// call fb cyclic
fbHoming.bCalibrationCam := bCalibrationCam;	
fbHoming.BufferMode := stHomingPrm.eBufferMode;
fbHoming.HomingMode := stHomingPrm.eHomingMode;
fbHoming.Options := stHomingPrm.stOptions;
fbHoming.Position := stHomingPrm.fPosition;
fbHoming(Axis := fbAxisRef);

// FB diagnostic and reset 
IF fbHoming.Execute AND NOT fbHoming.Busy THEN
	IF fbHoming.Error THEN
		nErrorId := fbHoming.ErrorID;
		M_SetLocalErrorS('Error axis homing: ErrId: ', TO_STRING(nErrorId));
	END_IF
	fbHoming.Execute := FALSE;
END_IF
		
// return if not in homing
IF eCommandExecute <> E_MotionCommand.eMotionCommand_home THEN
	RETURN;
END_IF

//aSClearText[0] := 'Antrieb GRST';	
//aSClearText := F_GetTranslatedTxtEx("engine home position", eLanguage);	
IF NOT fbHoming.Busy THEN
	fbHoming(Axis := fbAxisRef, Execute := TRUE);
	eCommandExecute := E_MotionCommand.eMotionCommand_none;
END_IF
END_ACTION

METHOD PRIVATE WfInitPositionOffset : BOOL
VAR_INPUT
END_VAR
VAR_INST
	fbAdsWriteOffset			:ADSWRITE;
	iStepSetPosOffset			:INT;
END_VAR


CASE iStepSetPosOffset OF
	
	0:
		// warte auf Trigger
		IF bStartInitPosOffset THEN
			// Position offset set
			bSetPositionOffsetDone := FALSE;
			// Current position offset value
			fCurrentPositionOffset := 0;			
			iStepSetPosOffset := 5;
		END_IF	
		
	5:
		IF fbAxisRef.NcToPlc.AxisId > 0 THEN
			iStepSetPosOffset := 6;
		ELSE
			M_SetLocalErrorEx(CONST.stTextListGlobal.stText_Comp.stText_Axis_FbError, F_CreateDynText("No Nc.AxisId!", 0));
		END_IF

	6:
		IF NOT Operational THEN
			iStepSetPosOffset := 10;
		ELSE
			M_SetLocalErrorEx(CONST.stTextListGlobal.stText_Comp.stText_Axis_FbError, F_CreateDynText("Axis is Operational. Please switch off axis!", 0));
		END_IF

	10:
		fbAdsWriteOffset.IDXGRP := 16#5000 + fbAxisRef.NcToPlc.AxisId;        (* Ind.Gr. f. AxisPara *)
		fbAdsWriteOffset.IDXOFFS := 16#7;
		fbAdsWriteOffset.LEN:= SIZEOF(fPosOffsetValToSet);
		fbAdsWriteOffset.SRCADDR:= ADR(fPosOffsetValToSet);
		fbAdsWriteOffset.WRITE:= TRUE;
		iStepSetPosOffset := 15;
   
    15:
        // 'wait until offset-parameter is handed over';
        IF NOT fbAdsWriteOffset.BUSY THEN
            IF fbAdsWriteOffset.ERRID = 0 THEN
				// Position offset set
				bSetPositionOffsetDone := TRUE;
				// Current position offset value
				fCurrentPositionOffset := fPosOffsetValToSet;
                iStepSetPosOffset := 100;
            ELSE
                M_SetLocalErrorEx(CONST.stTextListGlobal.stText_Comp.stText_Axis_FbError, F_CreateDynText("Error writing offset to NC.", 0));
				iStepSetPosOffset := 100;
            END_IF
        END_IF	
		

		// finish
	100:
		fbAdsWriteOffset.WRITE:= FALSE;
		bStartInitPosOffset := FALSE; // Finish
		fPosOffsetValToSet := 0;
		iStepSetPosOffset := 0;

END_CASE

fbAdsWriteOffset.PORT := 500;
fbAdsWriteOffset();
END_METHOD

ACTION WfJog:

/// Workflow jog axis

// call fb cyclic
fbjog.JogBackwards := stJogPrm.bJogBackwards AND Operational;
fbjog.JogForward := stJogPrm.bJogForward AND Operational;
fbjog.Acceleration := stJogPrm.fAcceleration;
fbjog.Deceleration := stJogPrm.fDeceleration;
fbjog.Jerk := stJogPrm.fJerk;
fbjog.Mode := stJogPrm.eMode;
fbjog.Position := stJogPrm.fPosition;
fbjog.Velocity := stJogPrm.fVelocity;
fbjog(Axis := fbAxisRef);

// reset jog F/B each cycle (stop's axis if Jog/JogEx method isn't called anymore)
stJogPrm.bJogBackwards := FALSE;
stJogPrm.bJogForward := FALSE;

// return if not in jog
IF eCommandExecute <> E_MotionCommand.eMotionCommand_jog THEN
	RETURN;
END_IF

// case of jog error
IF fbjog.Error  THEN
	nErrorId := fbjog.ErrorID;
	M_SetLocalErrorS('Error axis jogging: ErrId: ', TO_STRING(nErrorId));
END_IF		

eCommandExecute := E_MotionCommand.eMotionCommand_none;
END_ACTION

ACTION WfJogAcc:

/// Workflow jog axis acc

// call fb's cyclic
//fbJogAcc.Direction := MC_Current_Direction;
//IF stJogAccPrm.bJogForward OR stJogAccPrm.bJogBackwards THEN
fbJogAcc.Direction := SEL(stJogAccPrm.bJogForward, MC_Negative_Direction, MC_Positive_Direction);	
//END_IF
fbJogAcc.Acceleration := stJogAccPrm.fAcceleration;
fbJogAcc.Deceleration := stJogAccPrm.fDeceleration;
fbJogAcc.Jerk := stJogAccPrm.fJerk;
fbJogAcc.BufferMode := stJogAccPrm.eBufferMode;
fbJogAcc.Options := stJogAccPrm.stOptions;
fbJogAcc(Axis := fbAxisRef);

// FB diagnostic and reset 
IF fbJogAcc.Execute AND (NOT fbJogAcc.Busy OR fbJogAcc.InVelocity) THEN
	IF fbJogAcc.Error THEN
		nErrorId := fbJogAcc.ErrorID;
		M_SetLocalErrorS('Error axis jogging acceleration: ErrId: ', TO_STRING(nErrorId));
	END_IF
	fbJogAcc.Velocity := 0;
	fbJogAcc.Execute := FALSE;
END_IF

// measure jog time to capture speed at the according ramp positon
tonJogAcc.IN := stJogAccPrm.bJogForward OR stJogAccPrm.bJogBackwards;
tonJogAcc.PT := stJogAccPrm.tAccTime;
tonJogAcc();

// reset jog F/B each cycle (stop's axis if Jog/JogEx method isn't called anymore)
stJogAccPrm.bJogBackwards := FALSE;
stJogAccPrm.bJogForward := FALSE;

IF eCommandExecute <> E_MotionCommand.eMotionCommand_jogAcc THEN
	RETURN;
END_IF

// halt axis if jogAcc timer is disabled
IF NOT tonJogAcc.IN THEN
	fbJogAcc.Velocity := 0;
	eCommandExecute := E_MotionCommand.eMotionCommand_none;
	stHaltPrm.eBufferMode := MC_Aborting;
	stHaltPrm.fDeceleration := stJogAccPrm.fDeceleration;
	stHaltPrm.fJerk := stJogAccPrm.fJerk;
	stHaltPrm.stOptions := stJogAccPrm.stOptions;
	THIS^.HaltEx(stHaltPrm);	
END_IF

//aSClearText[0] := Concat2x('Antrieb Tippen Beschleunigung, Geschwindigkeit: ', LREAL_TO_STRING(fbJogAcc.Velocity));
//aSClearText := Concat2x(F_GetTranslatedTxtLib('type engine acceleration, acceleration: ', eLanguage), LREAL_TO_STRING(fbJogAcc.Velocity));
IF fbJogAcc.Velocity < stJogAccPrm.fFastSpeed AND NOT fbJogAcc.Busy THEN
	// ramp = Kx + d
	fbJogAcc.Velocity := (TIME_TO_LREAL(tonJogAcc.ET) * ((stJogAccPrm.fFastSpeed - stJogAccPrm.fSlowSpeed)/TIME_TO_LREAL(tonJogAcc.PT))) + stJogAccPrm.fSlowSpeed;
	// limit speed	
	fbJogAcc.Velocity := LIMIT(stJogAccPrm.fSlowSpeed, fbJogAcc.Velocity, stJogAccPrm.fFastSpeed);
	fbJogAcc(Axis := fbAxisRef, Execute := TRUE);	
END_IF
END_ACTION

ACTION WfMovAbs:

/// Workflow move axis abs

// call fb's cyclic
fbMovAbs1.Position := stMovAbsPrm.fPosition;
fbMovAbs1.Velocity := stMovAbsPrm.fVelocity;
fbMovAbs1.Acceleration := stMovAbsPrm.fAcceleration;
fbMovAbs1.Deceleration := stMovAbsPrm.fDeceleration;
fbMovAbs1.Jerk := stMovAbsPrm.fJerk;
fbMovAbs1.BufferMode := stMovAbsPrm.eBufferMode;
fbMovAbs1.Options := stMovAbsPrm.stOptions;
fbMovAbs1(Axis := fbAxisRef);

fbMovAbs2.Position := stMovAbsPrm.fPosition;
fbMovAbs2.Velocity := stMovAbsPrm.fVelocity;
fbMovAbs2.Acceleration := stMovAbsPrm.fAcceleration;
fbMovAbs2.Deceleration := stMovAbsPrm.fDeceleration;
fbMovAbs2.Jerk := stMovAbsPrm.fJerk;
fbMovAbs2.BufferMode := stMovAbsPrm.eBufferMode;
fbMovAbs2.Options := stMovAbsPrm.stOptions;
fbMovAbs2(Axis := fbAxisRef);

bMovAbsRdy := NOT (fbMovAbs1.Busy AND fbMovAbs2.Busy);

// FB diagnostic and reset 
IF fbMovAbs1.Execute AND NOT fbMovAbs1.Busy THEN
	IF fbMovAbs1.Error AND (fbMovAbs1.ErrorID <> 17022) THEN
		nErrorId := fbMovAbs1.ErrorID;
		M_SetLocalErrorS('engine positioning absolut (FB1): ErrId: ', TO_STRING(nErrorId));
	END_IF
	fbMovAbs1.Execute := FALSE;
END_IF
IF fbMovAbs2.Execute AND NOT fbMovAbs2.Busy THEN
	IF fbMovAbs2.Error AND (fbMovAbs2.ErrorID <> 17022) THEN
		nErrorId := fbMovAbs2.ErrorID;
		M_SetLocalErrorS('engine positioning absolut (FB2): ErrId: ', TO_STRING(nErrorId));
	END_IF
	fbMovAbs2.Execute := FALSE;
END_IF

// return if not in move abs
IF eCommandExecute <> E_MotionCommand.eMotionCommand_moveAbs THEN
	RETURN;
END_IF

//aSClearText[0] := 'Antrieb Positionierung Absolut';	
//aSClearText := F_GetTranslatedTxtLib('engine positioning absolut', eLanguage);
IF NOT fbMovAbs1.Busy THEN
	fbMovAbs1(Axis := fbAxisRef, Execute := TRUE);
	eCommandExecute := E_MotionCommand.eMotionCommand_none;
ELSIF NOT fbMovAbs2.Busy THEN
	fbMovAbs2(Axis := fbAxisRef, Execute := TRUE);
	eCommandExecute := E_MotionCommand.eMotionCommand_none;
ELSE
	nErrorId := 0;
	M_SetLocalError(F_CreateDynText("engine positioning absolut. No component ready", 0));
END_IF
END_ACTION

ACTION WfMovAdd:

/// Workflow move axis add

// call fb's cyclic
fbMovAdd1.Distance := stMovAddPrm.fDistance;
fbMovAdd1.Velocity := stMovAddPrm.fVelocity;
fbMovAdd1.Acceleration := stMovAddPrm.fAcceleration;
fbMovAdd1.Deceleration := stMovAddPrm.fDeceleration;
fbMovAdd1.Jerk := stMovAddPrm.fJerk;
fbMovAdd1.BufferMode := stMovAddPrm.eBufferMode;
fbMovAdd1.Options := stMovAddPrm.stOptions;
fbMovAdd1(Axis := fbAxisRef);

fbMovAdd2.Distance := stMovAddPrm.fDistance;
fbMovAdd2.Velocity := stMovAddPrm.fVelocity;
fbMovAdd2.Acceleration := stMovAddPrm.fAcceleration;
fbMovAdd2.Deceleration := stMovAddPrm.fDeceleration;
fbMovAdd2.Jerk := stMovAddPrm.fJerk;
fbMovAdd2.BufferMode := stMovAddPrm.eBufferMode;
fbMovAdd2.Options := stMovAddPrm.stOptions;
fbMovAdd2(Axis := fbAxisRef);

// FB diagnostic and reset 
IF fbMovAdd1.Execute AND NOT fbMovAdd1.Busy THEN
	IF fbMovAdd1.Error AND (fbMovAdd1.ErrorID <> 17022) THEN
		nErrorId := fbMovAdd1.ErrorID;
		M_SetLocalErrorS('engine positioning additive (FB1): ErrId: ', TO_STRING(nErrorId));
	END_IF
	fbMovAdd1.Execute := FALSE;
END_IF
IF fbMovAdd2.Execute AND NOT fbMovAdd2.Busy THEN
	IF fbMovAdd2.Error AND (fbMovAdd2.ErrorID <> 17022) THEN
		nErrorId := fbMovAdd2.ErrorID;
		M_SetLocalErrorS('engine positioning additive (FB2): ErrId: ', TO_STRING(nErrorId));
	END_IF
	fbMovAdd2.Execute := FALSE;
END_IF

// return if not in move add
IF eCommandExecute <> E_MotionCommand.eMotionCommand_moveAdd THEN
	RETURN;
END_IF

//aSClearText := F_GetTranslatedTxtLib('engine positioning additive', eLanguage);
IF NOT fbMovAdd1.Busy THEN
	fbMovAdd1(Axis := fbAxisRef, Execute := TRUE);
	eCommandExecute := E_MotionCommand.eMotionCommand_none;	
ELSIF NOT fbMovAdd2.Busy THEN
	fbMovAdd2(Axis := fbAxisRef, Execute := TRUE);
	eCommandExecute := E_MotionCommand.eMotionCommand_none;	
ELSE
	nErrorId := 0;
	M_SetLocalError(F_CreateDynText("engine positioning additive. No component ready", 0));
END_IF
END_ACTION

ACTION WfMovMod:

/// Workflow move axis mod

// call fb's cyclic
fbMovMod1.Position := stMovModPrm.fPosition;
fbMovMod1.Direction := stMovModPrm.eDirection;
fbMovMod1.Velocity := stMovModPrm.fVelocity;
fbMovMod1.Acceleration := stMovModPrm.fAcceleration;
fbMovMod1.Deceleration := stMovModPrm.fDeceleration;
fbMovMod1.Jerk := stMovModPrm.fJerk;
fbMovMod1.BufferMode := stMovModPrm.eBufferMode;
fbMovMod1.Options := stMovModPrm.stOptions;
fbMovMod1(Axis := fbAxisRef);

fbMovMod2.Position := stMovModPrm.fPosition;
fbMovMod2.Direction := stMovModPrm.eDirection;
fbMovMod2.Velocity := stMovModPrm.fVelocity;
fbMovMod2.Acceleration := stMovModPrm.fAcceleration;
fbMovMod2.Deceleration := stMovModPrm.fDeceleration;
fbMovMod2.Jerk := stMovModPrm.fJerk;
fbMovMod2.BufferMode := stMovModPrm.eBufferMode;
fbMovMod2.Options := stMovModPrm.stOptions;
fbMovMod2(Axis := fbAxisRef);

// FB diagnostic and reset 
IF fbMovMod1.Execute AND NOT fbMovMod1.Busy THEN
	IF fbMovMod1.Error AND (fbMovMod1.ErrorID <> 17022) THEN
		nErrorId := fbMovMod1.ErrorID;
		M_SetLocalErrorS('engine positioning modulo (FB1): ErrId: ', TO_STRING(nErrorId));
	END_IF
	fbMovMod1.Execute := FALSE;
END_IF
IF fbMovMod2.Execute AND NOT fbMovMod2.Busy THEN
	IF fbMovMod2.Error AND (fbMovMod2.ErrorID <> 17022) THEN
		nErrorId := fbMovMod2.ErrorID;
		M_SetLocalErrorS('engine positioning modulo (FB2): ErrId: ', TO_STRING(nErrorId));
	END_IF
	fbMovMod2.Execute := FALSE;
END_IF

// return if not in move rel
IF eCommandExecute <> E_MotionCommand.eMotionCommand_moveMod THEN
	RETURN;
END_IF

//aSClearText[0] := 'Antrieb Positionierung Modulo';	
//aSClearText := F_GetTranslatedTxtLib('engine positioning modulo', eLanguage);	
IF NOT fbMovMod1.Busy THEN
	fbMovMod1(Axis := fbAxisRef, Execute := TRUE);
	eCommandExecute := E_MotionCommand.eMotionCommand_none;
ELSIF NOT fbMovMod2.Busy THEN
	fbMovMod2(Axis := fbAxisRef, Execute := TRUE);
	eCommandExecute := E_MotionCommand.eMotionCommand_none;
ELSE
	nErrorId := 0;
	M_SetLocalError(F_CreateDynText("engine positioning modulo. No component ready", 0));
END_IF
END_ACTION

ACTION WfMovRel:

/// Workflow move axis rel

// call fb's cyclic
fbMovRel1.Distance := stMovRelPrm.fDistance;
fbMovRel1.Velocity := stMovRelPrm.fVelocity;
fbMovRel1.Acceleration := stMovRelPrm.fAcceleration;
fbMovRel1.Deceleration := stMovRelPrm.fDeceleration;
fbMovRel1.Jerk := stMovRelPrm.fJerk;
fbMovRel1.BufferMode := stMovRelPrm.eBufferMode;
fbMovRel1.Options := stMovRelPrm.stOptions;
fbMovRel1(Axis := fbAxisRef);

fbMovRel2.Distance := stMovRelPrm.fDistance;
fbMovRel2.Velocity := stMovRelPrm.fVelocity;
fbMovRel2.Acceleration := stMovRelPrm.fAcceleration;
fbMovRel2.Deceleration := stMovRelPrm.fDeceleration;
fbMovRel2.Jerk := stMovRelPrm.fJerk;
fbMovRel2.BufferMode := stMovRelPrm.eBufferMode;
fbMovRel2.Options := stMovRelPrm.stOptions;
fbMovRel2(Axis := fbAxisRef);

// FB diagnostic and reset 
IF fbMovRel1.Execute AND NOT fbMovRel1.Busy THEN
	IF fbMovRel1.Error AND (fbMovRel1.ErrorID <> 17022) THEN
		nErrorId := fbMovRel1.ErrorID;
		M_SetLocalErrorS('engine positioning relativ (FB1): ErrId: ', TO_STRING(nErrorId));
	END_IF
	fbMovRel1.Execute := FALSE;
END_IF
IF fbMovRel2.Execute AND NOT fbMovRel2.Busy THEN
	IF fbMovRel2.Error AND (fbMovRel2.ErrorID <> 17022) THEN
		nErrorId := fbMovRel2.ErrorID;
		M_SetLocalErrorS('engine positioning relativ (FB2): ErrId: ', TO_STRING(nErrorId));
	END_IF
	fbMovRel2.Execute := FALSE;
END_IF

// return if not in move rel
IF eCommandExecute <> E_MotionCommand.eMotionCommand_moveRel THEN
	RETURN;
END_IF

//aSClearText := F_GetTranslatedTxtLib('engine positioning relativ', eLanguage);
IF NOT fbMovRel1.Busy THEN
	fbMovRel1(Axis := fbAxisRef, Execute := TRUE);
	eCommandExecute := E_MotionCommand.eMotionCommand_none;	
ELSIF NOT fbMovRel2.Busy THEN
	fbMovRel2(Axis := fbAxisRef, Execute := TRUE);
	eCommandExecute := E_MotionCommand.eMotionCommand_none;	
ELSE
	nErrorId := 0;
	M_SetLocalError(F_CreateDynText("engine positioning relativ. No component ready", 0));
END_IF
END_ACTION

ACTION WfMovVel:

/// Workflow move axis vel

// call fb's cyclic
fbMovVel1.Velocity := stMovVelPrm.fVelocity;
fbMovVel1.Direction := stMovVelPrm.eDirection;
fbMovVel1.Acceleration := stMovVelPrm.fAcceleration;
fbMovVel1.Deceleration := stMovVelPrm.fDeceleration;
fbMovVel1.Jerk := stMovVelPrm.fJerk;
fbMovVel1.BufferMode := stMovVelPrm.eBufferMode;
fbMovVel1.Options := stMovVelPrm.stOptions;
fbMovVel1(Axis := fbAxisRef);

fbMovVel2.Velocity := stMovVelPrm.fVelocity;
fbMovVel2.Direction := stMovVelPrm.eDirection;
fbMovVel2.Acceleration := stMovVelPrm.fAcceleration;
fbMovVel2.Deceleration := stMovVelPrm.fDeceleration;
fbMovVel2.Jerk := stMovVelPrm.fJerk;
fbMovVel2.BufferMode := stMovVelPrm.eBufferMode;
fbMovVel2.Options := stMovVelPrm.stOptions;
fbMovVel2(Axis := fbAxisRef);

// FB diagnostic and reset 
IF fbMovVel1.Execute AND NOT fbMovVel1.Busy THEN
	IF fbMovVel1.Error AND (fbMovVel1.ErrorID <> 17022) THEN
		nErrorId := fbMovVel1.ErrorID;
		M_SetLocalErrorS('engine constant velocity (FB1): ErrId: ', TO_STRING(nErrorId));
	END_IF
	fbMovVel1.Execute := FALSE;
END_IF
IF fbMovVel2.Execute AND NOT fbMovVel2.Busy THEN
	IF fbMovVel2.Error AND (fbMovVel2.ErrorID <> 17022) THEN
		nErrorId := fbMovVel2.ErrorID;
		M_SetLocalErrorS('engine constant velocity (FB2): ErrId: ', TO_STRING(nErrorId));
	END_IF
	fbMovVel2.Execute := FALSE;
END_IF

// return if other command active
IF eCommandExecute <> E_MotionCommand.eMotionCommand_moveVel THEN
	RETURN;
END_IF

//aSClearText[0] := 'Antrieb Konstante Geschwindigkeit';
//aSClearText := F_GetTranslatedTxtLib('engine constant velocity', eLanguage);				
IF NOT fbMovVel1.Busy THEN
	fbMovVel1(Axis := fbAxisRef, Execute := TRUE);
	eCommandExecute := E_MotionCommand.eMotionCommand_none;
ELSIF NOT fbMovVel2.Busy THEN
	fbMovVel2(Axis := fbAxisRef, Execute := TRUE);
	eCommandExecute := E_MotionCommand.eMotionCommand_none;
ELSE
	nErrorId := 0;
	M_SetLocalError(F_CreateDynText("engine constant velocity. No Component ready", 0));
END_IF
END_ACTION

ACTION WfPower:

/// Workflow power axis

tonAutoPowerOff(IN := bEnable AND bEnableAutoPowerOff AND fbAxisRef.Status.NotMoving AND NOT fbAxisRef.Status.Error AND 
					  (eCommandRequest = eMotionCommand_none OR eCommandRequest = eMotionCommand_reset OR eCommandRequest = eMotionCommand_setPos) AND
					  (eCommandExecute = eMotionCommand_none OR eCommandExecute = eMotionCommand_reset OR eCommandExecute = eMotionCommand_setPos),
				PT := stDefaultPrm.stGeneralPrm.tAutoPowerOffDelay);

tonEnable(IN:=bEnable,PT := tEnableTime);
				
fbPower.Enable := tonEnable.Q AND NOT tonAutoPowerOff.Q;
fbPower.Enable_Negative := bEnableNeg;
fbPower.Enable_Positive := bEnablePos;
fbPower.Override := SEL(bHoldActiv,fSetOverride,0);
fbPower(BufferMode := MC_Aborting, Axis := fbAxisRef);

// ext. fan control
IF stIn.iMotorTemperature >= stDefaultPrm.stGeneralPrm.iExtFanThreshold THEN
	stOut.bExternalFan := TRUE;
ELSIF stIn.iMotorTemperature < (stDefaultPrm.stGeneralPrm.iExtFanThreshold - 50) THEN // hysteresis 5°C
	stOut.bExternalFan := FALSE;
END_IF

posPowerError(CLK := eState <> E_ComponentState.eComponentState_error AND fbPower.Error);
IF posPowerError.Q THEN
	nErrorId := fbPower.ErrorID;
	M_SetLocalErrorS('Axis power error: ErrId: ', TO_STRING(nErrorId));
END_IF
END_ACTION

ACTION WfReset:

/// Workflow resetting

// call FB cyclic
fbReset(Axis:= fbAxisRef);

// FB diagnostic and reset 
IF fbReset.Execute AND NOT fbReset.Busy THEN
	IF fbReset.Error THEN			
		nErrorId := fbReset.ErrorID;
		M_SetLocalErrorS('Error on engine reset: ErrId: ', TO_STRING(nErrorId));
	END_IF
	fbReset.Execute := FALSE;
END_IF

// force MC reset
IF eCommandExecute = eMotionCommand_resetMc THEN
	//aSClearText[0] := 'Start Antrieb MC Reset';
	//aSClearText := F_GetTranslatedTxtEx("Start engine MC reset", eLanguage);
	IF NOT fbReset.Busy THEN
		fbReset(Axis := fbAxisRef, Execute := TRUE);
		eCommandExecute := E_MotionCommand.eMotionCommand_none;
	END_IF
END_IF

// return if other command active
IF eCommandExecute <> E_MotionCommand.eMotionCommand_reset THEN
	RETURN;
END_IF

IF eAxisType = E_AxisType.AX5xxx THEN
	// reset ax5000
	//aSClearText := F_GetTranslatedTxtEx("Start engine reset", eLanguage);
	IF NOT fbAX5xxxDiag.Busy THEN
		fbAX5xxxDiag.Reset := fbAxisRef.Status.Error;
		eCommandExecute := E_MotionCommand.eMotionCommand_none;
		eState := E_ComponentState.eComponentState_ready;
	END_IF

// Bosch Indradrive
ELSIF eAxisType = E_AxisType.Bosch_IndradriveEc THEN
	// reset indradrive
	//aSClearText := F_GetTranslatedTxtEx("Start engine reset", eLanguage);
	IF NOT fbIndraDrvDiag.bBusy THEN
		fbIndraDrvDiag.bReset := fbAxisRef.Status.Error;
		eCommandExecute := E_MotionCommand.eMotionCommand_none;
		eState := E_ComponentState.eComponentState_ready;
	END_IF

ELSE
	// reset sequence of default axis types
	//aSClearText := F_GetTranslatedTxtEx("Start engine reset", eLanguage);
	IF NOT fbReset.Busy THEN
		fbReset(Axis := fbAxisRef, Execute := fbAxisRef.Status.Error);
		eCommandExecute := E_MotionCommand.eMotionCommand_none;
		eState := E_ComponentState.eComponentState_ready;
	END_IF
END_IF
END_ACTION

ACTION WfSetPos:

/// Workflow set position

// call fb cyclic
fbSetPos.Position := stSetPosPrm.fPosition;
fbSetPos.Mode := stSetPosPrm.bMode;
fbSetPos.Options := stSetPosPrm.stOptions;
fbSetPos(Axis := fbAxisRef);

// FB diagnostic and reset 
IF fbSetPos.Execute AND NOT fbSetPos.Busy THEN
	IF fbSetPos.Error THEN			
		nErrorId := fbSetPos.ErrorID;
		M_SetLocalErrorS('Error set engine position: ErrId: ', TO_STRING(nErrorId));
	END_IF
	fbSetPos.Execute := FALSE;
END_IF

// return if other command active	
IF eCommandExecute <> E_MotionCommand.eMotionCommand_setPos THEN
	RETURN;
END_IF

//aSClearText := F_GetTranslatedTxtLib('Set engine position', eLanguage);		
IF NOT fbSetPos.Busy THEN
	fbSetPos(Axis := fbAxisRef, Execute := TRUE);
	eCommandExecute := E_MotionCommand.eMotionCommand_none;
END_IF
END_ACTION

ACTION WfSoE:
// SoE commands
CASE stSoE.eCmd OF
	
	E_SoECommand.eSoECommand_writeIndraDrvPos:
		CASE stSoE.nStep OF
			0:	
				stSoE.fRealValue := (stSoE.fRealValue * 10000);
				diTempVal := REAL_TO_DINT(stSoE.fRealValue);
				stSoE.fbSoEWrite(
					Axis    := fbAxisRef,
					Idn := S_0_IDN + 52, 				// S-0-0052, Referenzmaß 1
					Element := EC_SOE_ELEMENT_VALUE,
					pSrcBuf  := ADR(diTempVal),	// Position
					BufLen   := SIZEOF(diTempVal),
					//Password := Password,				// Password   : ST_SoE_String;
					Execute  := TRUE,
					Timeout  := DEFAULT_ADS_TIMEOUT);				
				IF NOT stSoE.fbSoEWrite.Busy THEN
					IF stSoE.fbSoEWrite.Error THEN
						eState := E_ComponentState.eComponentState_error;
						nErrorID := stSoE.fbSoEWrite.AdsErrId;
						M_SetLocalError(F_CreateDynText(TO_WSTRING(Concat4('SoEWrite error, AdsErrId: ', UINT_TO_STRING(stSoE.fbSoEWrite.AdsErrId), ', SercosErrId: ', UINT_TO_STRING(stSoE.fbSoEWrite.SercosErrId))), 0));
						stSoE.nStep := 0;
						stSoE.eCmd := E_SoECommand.eSoECommand_none;
					ELSE
						stSoE.nStep := 10;
					END_IF
					stSoE.fbSoEWrite(Axis := fbAxisRef, Execute := FALSE);
				END_IF
				
			10:	stSoE.fbSoECmd(
					Axis    := fbAxisRef,
					Execute := TRUE,
					Timeout := DEFAULT_ADS_TIMEOUT,
					Idn     := S_0_IDN + 447);			// C0300 Kommando Absolutmaß setzen		P_0_IDN + 12
				IF NOT stSoE.fbSoECmd.Busy THEN
					IF stSoE.fbSoECmd.Error THEN
						eState := E_ComponentState.eComponentState_error;
						nErrorID := stSoE.fbSoEWrite.AdsErrId;
						M_SetLocalError(F_CreateDynText(TO_WSTRING(Concat4('SoECmd error, AdsErrId: ', UINT_TO_STRING(stSoE.fbSoECmd.AdsErrId), ', SercosErrId: ', UINT_TO_STRING(stSoE.fbSoECmd.SercosErrId))), 0));
					END_IF
					stSoE.fbSoECmd(Axis := fbAxisRef, Execute := FALSE);
					stSoE.nStep := 0;
					stSoE.eCmd := E_SoECommand.eSoECommand_none;
				END_IF
				
		END_CASE
		
END_CASE
END_ACTION

ACTION WfStop:

/// Workflow stopping

// call fb cyclic
fbStop.Deceleration := stStopPrm.fDeceleration;
fbStop.Jerk := stStopPrm.fJerk;
fbStop.Options := stStopPrm.stOptions;
fbStop(Axis := fbAxisRef);

// FB diagnostic and reset
IF fbStop.Execute THEN
	IF fbStop.Error THEN			
		nErrorId := fbStop.ErrorID;
		M_SetLocalErrorS('Error stopping axis: ErrId: ', TO_STRING(nErrorId));
	END_IF
	fbStop.Execute := FALSE;
END_IF

// return if other command active
IF eCommandExecute <> E_MotionCommand.eMotionCommand_stop THEN
	RETURN;
END_IF

//aSClearText[0] := 'Antrieb Stoppen';
//aSClearText := F_GetTranslatedTxtLib('stop the engine ', eLanguage);
fbStop(Axis := fbAxisRef, Execute := TRUE);

// stop command is not auto reset -> ext. reset needed!

//IF fbAxisRef.Status.StandStill AND fbStop.Done AND NOT fbStop.Busy THEN
	eCommandExecute := E_MotionCommand.eMotionCommand_none;
//END_IF
END_ACTION

ACTION WfTorqCtrl:

/// Workflow torque control
stTorqCtrlPrm.stOptions.ManualTorqueStartValue := fbAxisRef.NcToPlc.ActTorque;
stTorqCtrlPrm.stOptions.EnableManualTorqueStartValue := TRUE;

// call fb cyclic
fbTorqueControl.Torque := stTorqCtrlPrm.fTorque;
fbTorqueControl.TorqueRamp := stTorqCtrlPrm.fTorqueRamp;
fbTorqueControl.VelocityLimitHigh := stTorqCtrlPrm.fVelocityLimitHigh;
fbTorqueControl.VelocityLimitLow := stTorqCtrlPrm.fVelocityLimitLow;
fbTorqueControl.ContinuousUpdate := stTorqCtrlPrm.bContinuousUpdate;
fbTorqueControl.Relative := stTorqCtrlPrm.bRelative;
fbTorqueControl.BufferMode := stTorqCtrlPrm.eBufferMode;
fbTorqueControl.Options := stTorqCtrlPrm.stOptions;
fbTorqueControl(Axis := fbAxisRef);

// FB diagnostic and reset 
IF fbTorqueControl.Execute AND NOT fbTorqueControl.Busy THEN
	IF fbTorqueControl.Error AND (fbTorqueControl.ErrorID <> 17022) THEN
		nErrorId := fbTorqueControl.ErrorID;
		M_SetLocalErrorS('engine torque control: ErrId: ', TO_STRING(nErrorId));
	END_IF
	fbTorqueControl.Execute := FALSE;
END_IF

// return if not in torque control
IF eCommandExecute <> E_MotionCommand.eMotionCommand_torqCtrl THEN
	RETURN;
END_IF

//IF NOT fbTorqueControl.Busy THEN
	fbTorqueControl(Axis := fbAxisRef, ContinuousUpdate := stTorqCtrlPrm.bContinuousUpdate, Execute := TRUE);
	eCommandExecute := E_MotionCommand.eMotionCommand_none;
//ELSE
//	nErrorId := 0;
//	M_SetLocalError(F_CreateDynText("engine torque control. Component not ready", 0));
//END_IF
END_ACTION

END_FUNCTION_BLOCK

// ---- POUs/MAIN_Fast.TcPOU
PROGRAM MAIN_Fast
VAR_INPUT
END_VAR
VAR
END_VAR
VAR_OUTPUT	
END_VAR

// fast stuff here..

fbModul001.M_Fast();

END_PROGRAM

// ---- POUs/HMI/Provider/HwHmi/FB_HMI_PROVIDER_HW.TcPOU
FUNCTION_BLOCK FB_HMI_PROVIDER_HW EXTENDS FB_HMI_PROVIDER_BASE
VAR
	stIn		: REFERENCE TO HMI_PROVIDER_HW_IN;
	stOut		: REFERENCE TO HMI_PROVIDER_HW_OUT;
	bLedTest	: BOOL;
	
	nSelStation : E_Station;
	bAlternativ : BOOL;	
	bJog : BOOL;
	bSpeed : BOOL;

	
END_VAR

METHOD M_EuchnerToPLC : BOOL
VAR_INST		
	fbSelection				:FB_TON_RMTH;
	fbAlt					:FB_TON_RMTH;
	fbJog					:FB_TON_RMTH;
	fbSpeed					:FB_TON_RMTH;
	
	rtrigJog01				:R_TRIG;
	rtrigJog02				:R_TRIG;
	rtrigReset				:R_TRIG;
	
	nNewSelection			: INT;
END_VAR
fbSelection(IN := stIn.stP51A_S1HandBs.bSelect01 OR stIn.stP51A_S1HandBs.bSelect02 OR stIn.stP51A_S1HandBs.bSelect03 OR stIn.stP51A_S1HandBs.bSelect04 OR stIn.stP51A_S1HandBs.bSelect05 OR stIn.stP51A_S1HandBs.bSelect06 , PT:= T#50MS);	//Selection
fbAlt(IN := stIn.stP51A_S1HandBs.bAlt, PT:= T#50MS);	//Selection

fbJog(IN := stIn.stP51A_S1HandBs.bJog, PT:= T#50MS, Qr=> bJog);	//Selection
stIn.stSt010.bJog := stIn.stSt020.bJog := stIn.stSt030.bJog := stIn.stSt040.bJog := bJog;

fbSpeed(IN := stIn.stP51A_S1HandBs.bDistance, PT:= T#50MS);	//Selection

IF fbSpeed.Qr THEN
	bSpeed := NOT bSpeed;
END_IF

IF fbJog.Qr THEN
	bSpeed := FALSE;	
END_IF

stIn.stSt010.bSpeed := stIn.stSt020.bSpeed := stIn.stSt030.bSpeed := stIn.stSt040.bSpeed := bSpeed;

// Umschalten Station
IF fbSelection.Qr THEN
	bAlternativ := FALSE;
	IF stIn.stP51A_S1HandBs.bSelect01 THEN
		nNewSelection := E_Station.eStation_ST010_OvenA;
	ELSIF stIn.stP51A_S1HandBs.bSelect02 THEN
		nNewSelection := E_Station.eStation_ST020_OvenB;		
	ELSIF stIn.stP51A_S1HandBs.bSelect03 THEN
		nNewSelection := E_Station.eStation_ST030_Handling;		
	ELSIF stIn.stP51A_S1HandBs.bSelect04 THEN
		nNewSelection := E_Station.eStation_ST040_Storage;		
	ELSIF stIn.stP51A_S1HandBs.bSelect05 THEN
		nNewSelection := E_Station.eStation_ST050_Mould;		
	ELSIF stIn.stP51A_S1HandBs.bSelect06 THEN
		nNewSelection := E_Station.eStation_none;		
	END_IF
	
	IF nNewSelection = nSelStation THEN
		nSelStation := E_Station.eStation_none;
	ELSE
		nSelStation := nNewSelection;
	END_IF	
	
END_IF


// Umschalten auf Alternativ
IF fbAlt.Qr THEN
	bAlternativ := NOT bAlternativ;
END_IF
rtrigJog01(CLK := stIn.stP51A_S1HandBs.bLeft OR stIn.stP51A_S1HandBs.bRight);
rtrigJog02(CLK := stIn.stP51A_S1HandBs.bDown OR stIn.stP51A_S1HandBs.bUp);
rtrigReset(CLK := );

// Stationsfunktionen
CASE nSelStation OF
	

	eStation_none:  stIn.stM001.bQuit := stIn.stP51A_S1HandBs.bReset;

	
	eStation_ST010_OvenA: 	//stIn.stSt010.bManual := stIn.stP51A_S1HandBs.bReset;	
		stIn.stSt010.bQuit := stIn.stP51A_S1HandBs.bReset;

		// set up index	
		IF NOT bAlternativ THEN
			stOut.stP51A_S1HandBs.bLedLeft := TRUE;
			stOut.stP51A_S1HandBs.bLedRight := TRUE;	
			stIn.stSt010.bJogCh1Inside := stIn.stP51A_S1HandBs.bLeft;
	   		stIn.stSt010.bJogCh1Ouside := stIn.stP51A_S1HandBs.bRight;	
			IF rtrigJog01.Q THEN
				stIn.arrStStation[E_Station.eStation_ST010_OvenA].stManual.diSelectedObjectIndex := fbSt010OvenA.fbAxisCh1Ui.diObjectIndex;			
				bRequestManualControl := TRUE;
			END_IF					
		ELSE
			stOut.stP51A_S1HandBs.bLedLeft := TRUE;
			stOut.stP51A_S1HandBs.bLedRight := TRUE;
			stIn.stSt010.bJogCh2Inside := stIn.stP51A_S1HandBs.bLeft;
	   		stIn.stSt010.bJogCh2Ouside := stIn.stP51A_S1HandBs.bRight;	
			IF rtrigJog01.Q THEN
				stIn.arrStStation[E_Station.eStation_ST010_OvenA].stManual.diSelectedObjectIndex := fbSt010OvenA.fbAxisCh2Ui.diObjectIndex;
				bRequestManualControl := TRUE;
			END_IF
		END_IF
		
		stOut.stP51A_S1HandBs.bLedUp := TRUE;
		stOut.stP51A_S1HandBs.bLedDown := TRUE;
		stIn.stSt010.bJogUp := stIn.stP51A_S1HandBs.bUp;
		stIn.stSt010.bJogDown := stIn.stP51A_S1HandBs.bDown;
		IF rtrigJog02.Q THEN
			stIn.arrStStation[E_Station.eStation_ST010_OvenA].stManual.diSelectedObjectIndex := fbSt010OvenA.fbAxisUi.diObjectIndex;
			bRequestManualControl := TRUE;
		END_IF		
	
	eStation_ST020_OvenB: 	//stIn.stSt020.bManual := stIn.stP51A_S1HandBs.bReset;
		stIn.stSt020.bQuit := stIn.stP51A_S1HandBs.bReset;

		IF NOT bAlternativ THEN
			stOut.stP51A_S1HandBs.bLedLeft := TRUE;
			stOut.stP51A_S1HandBs.bLedRight := TRUE;	
			stIn.stSt020.bJogCh1Inside := stIn.stP51A_S1HandBs.bLeft;
	   		stIn.stSt020.bJogCh1Ouside := stIn.stP51A_S1HandBs.bRight;	
			IF rtrigJog01.Q THEN
				stIn.arrStStation[E_Station.eStation_ST020_OvenB].stManual.diSelectedObjectIndex := fbSt020OvenB.fbAxisCh1Ui.diObjectIndex;
				bRequestManualControl := TRUE;
			END_IF					
		ELSE
			stOut.stP51A_S1HandBs.bLedLeft := TRUE;
			stOut.stP51A_S1HandBs.bLedRight := TRUE;
			stIn.stSt020.bJogCh2Inside := stIn.stP51A_S1HandBs.bLeft;
	   		stIn.stSt020.bJogCh2Ouside := stIn.stP51A_S1HandBs.bRight;	
			IF rtrigJog01.Q THEN
				stIn.arrStStation[E_Station.eStation_ST020_OvenB].stManual.diSelectedObjectIndex := fbSt020OvenB.fbAxisCh2Ui.diObjectIndex;
				bRequestManualControl := TRUE;
			END_IF
		END_IF
		
		stOut.stP51A_S1HandBs.bLedUp := TRUE;
		stOut.stP51A_S1HandBs.bLedDown := TRUE;
		stIn.stSt020.bJogUp := stIn.stP51A_S1HandBs.bUp;
		stIn.stSt020.bJogDown := stIn.stP51A_S1HandBs.bDown;
		IF rtrigJog02.Q THEN
			stIn.arrStStation[E_Station.eStation_ST020_OvenB].stManual.diSelectedObjectIndex := fbSt020OvenB.fbAxisUi.diObjectIndex;
			bRequestManualControl := TRUE;
		END_IF	
	
	
	eStation_ST030_Handling: 	//stIn.stSt030.bManual := stIn.stP51A_S1HandBs.bReset;
		stIn.stSt030.bQuit := stIn.stP51A_S1HandBs.bReset;
	
		IF NOT bAlternativ THEN
			stOut.stP51A_S1HandBs.bLedLeft := TRUE;
			stOut.stP51A_S1HandBs.bLedRight := TRUE;
			stIn.stSt030.bJogXN := stIn.stP51A_S1HandBs.bLeft;
	   		stIn.stSt030.bJogXP := stIn.stP51A_S1HandBs.bRight;	
			IF rtrigJog01.Q THEN
				stIn.arrStStation[E_Station.eStation_ST030_Handling].stManual.diSelectedObjectIndex := fbSt030Handling.fbAxisXUi.diObjectIndex;
				bRequestManualControl := TRUE;
			END_IF	
			
			stOut.stP51A_S1HandBs.bLedUp := TRUE;
			stOut.stP51A_S1HandBs.bLedDown := TRUE;	
			stIn.stSt030.bJogYN := stIn.stP51A_S1HandBs.bDown;
	   		stIn.stSt030.bJogYP := stIn.stP51A_S1HandBs.bUp;
			IF rtrigJog02.Q THEN
				stIn.arrStStation[E_Station.eStation_ST030_Handling].stManual.diSelectedObjectIndex := fbSt030Handling.fbAxisYUi.diObjectIndex;
				bRequestManualControl := TRUE;
			END_IF	
	
		ELSE
			stOut.stP51A_S1HandBs.bLedLeft := TRUE;
			stOut.stP51A_S1HandBs.bLedRight := TRUE;
			stIn.stSt030.bJogZN := stIn.stP51A_S1HandBs.bLeft;
			stIn.stSt030.bJogZP := stIn.stP51A_S1HandBs.bRight;
			IF rtrigJog01.Q THEN
				stIn.arrStStation[E_Station.eStation_ST030_Handling].stManual.diSelectedObjectIndex := fbSt030Handling.fbAxisZUi.diObjectIndex;
				bRequestManualControl := TRUE;
			END_IF	
					
			stOut.stP51A_S1HandBs.bLedUp := FALSE;
			stOut.stP51A_S1HandBs.bLedDown := FALSE;
			
		END_IF		
		
	eStation_ST040_Storage: 	//stIn.stSt040.bManual := stIn.stP51A_S1HandBs.bReset;
		stIn.stSt040.bQuit := stIn.stP51A_S1HandBs.bReset;

		stOut.stP51A_S1HandBs.bLedLeft := FALSE;
		stOut.stP51A_S1HandBs.bLedRight := FALSE;	
	
		IF NOT bAlternativ THEN
			stOut.stP51A_S1HandBs.bLedUp := TRUE;
			stOut.stP51A_S1HandBs.bLedDown := TRUE;
			stIn.stSt040.bJog01Down := stIn.stP51A_S1HandBs.bDown;
	   		stIn.stSt040.bJog01Up := stIn.stP51A_S1HandBs.bUp;
			IF rtrigJog02.Q THEN
				stIn.arrStStation[E_Station.eStation_ST040_Storage].stManual.diSelectedObjectIndex := fbSt040Storage.fbAxis1Ui.diObjectIndex;
				bRequestManualControl := TRUE;
			END_IF					
		ELSE
			stOut.stP51A_S1HandBs.bLedUp := TRUE;
			stOut.stP51A_S1HandBs.bLedDown := TRUE;
			stIn.stSt040.bJog02Down := stIn.stP51A_S1HandBs.bDown;
	   		stIn.stSt040.bJog02Up := stIn.stP51A_S1HandBs.bUp;
			IF rtrigJog02.Q THEN
				stIn.arrStStation[E_Station.eStation_ST040_Storage].stManual.diSelectedObjectIndex := fbSt040Storage.fbAxis2Ui.diObjectIndex;
				bRequestManualControl := TRUE;
			END_IF
		END_IF
				

END_CASE




// chk control request, e.g.: watch for changes --> stIn..bJog.. (for continuous jog only!)
END_METHOD

METHOD PRIVATE M_HmiToPlc : BOOL
VAR_INST
	rtrigDoorP30A,
	rtrigDoorOpnP50A,
	rtrigDoorClsP50A,
	rtrigVorwHaerten,
	rtrigVorwAnlassen,
	rtrigAutoKorrS1,
	rtrigAutoKorrS2,
	rtrigAutoKorrS3,
	rtrigJog : R_TRIG;
END_VAR
/// general
stIn.stMain.stButton_Start.bClick := // stIn.stP10A_OvenA.bAutoOn OR	// Automatik Ein; LDT-GN, 1DI-NO, 1DO; +P30A-21SJ2
									 stIn.stP50A_Haupt.bAutoOn;				// Automatik Ein, LDT-GN, 1DI-NO, 1DO, BMK: +P50A-21SJ2

stIn.stMain.stButton_Stop.bClick := stIn.stP50A_Haupt.bAutoOff;// OR			// Automatik Aus, DT-RD, 1DI-NO, BMK: +P50A-21SJ3
									//stIn.stP10B_OvenB.bAutoOff;		// Automatik Aus; DT-RD, 1DI-NO; P10B-1SG2

//stIn.stMain.stButton_Home.bClick := stIn.bTaste_GRST;
//stIn.stMain.stButton_Step.bClick := stIn.bTaste_Tipp;
stIn.stMain.stButton_Reset.bClick := stIn.stP50A_Haupt.bEsQuit;// OR
									 //stIn.stP10A_OvenA.bReset;

//stIn.stMain.stButton_OPM_Manual.bClick := stIn.bTaste_BA_Hand;
//stIn.stMain.stButton_OPM_Step.bClick := stIn.bTaste_BA_Einricht;
//stIn.stMain.stButton_OPM_Auto.bClick := stIn.bTaste_BA_Auto;
stIn.stSafety.bQuitSafety := stIn.stP50A_Haupt.bEsQuit; // OR			// Not-Halt Quittieren, LDT-BU, 1DI-NO, 1DO, BMK: +P50A-21SJ1
								//stIn.stP10A_OvenA.bReset;	// Reset Not-Halt; LDT-BU, 1DI-NO, 1DO; +P30A-21SJX
END_METHOD

METHOD PUBLIC M_Init : BOOL
VAR
END_VAR
eProvider := E_HMI_PROVIDER.eHmiProvider_HW;
//ILog := SERVICES.ILog;
M_SetReferences(HMI.stHmiHw.stIn, HMI.stHmiHw.stOut);

//aSClearText[EN] := 'HMI init done.';
M_Init := SUPER^.M_Init();
END_METHOD

METHOD M_PlcToEuchner : BOOL
VAR_INPUT
END_VAR
stOut.stP51A_S1HandBs.bLedSelect01 := FALSE;
stOut.stP51A_S1HandBs.bLedSelect02 := FALSE;
stOut.stP51A_S1HandBs.bLedSelect03 := FALSE;
stOut.stP51A_S1HandBs.bLedSelect04 := FALSE;
stOut.stP51A_S1HandBs.bLedSelect05 := FALSE;
stOut.stP51A_S1HandBs.bLedSelect06 := FALSE;

CASE nSelStation OF
	
	0: stOut.stP51A_S1HandBs.bLedSelect01 := SEL(plant.fbSt010OvenA.State > eComponentState_running, TRUE, Statics.stPulse.bToggle1000ms);
	   stOut.stP51A_S1HandBs.bLedSelect02 := SEL(plant.fbSt020OvenB.State > eComponentState_running, TRUE, Statics.stPulse.bToggle1000ms);
	   stOut.stP51A_S1HandBs.bLedSelect03 := SEL(plant.fbSt030Handling.State > eComponentState_running, TRUE, Statics.stPulse.bToggle1000ms);
	   stOut.stP51A_S1HandBs.bLedSelect04 := SEL(plant.fbSt040Storage.State > eComponentState_running, TRUE, Statics.stPulse.bToggle1000ms);
	   stOut.stP51A_S1HandBs.bLedSelect05 := SEL(plant.fbSt050Mould.State > eComponentState_running, TRUE, Statics.stPulse.bToggle1000ms);

	1: stOut.stP51A_S1HandBs.bLedSelect01 := SEL(plant.fbSt010OvenA.State > eComponentState_running, TRUE, Statics.stPulse.bToggle1000ms);
	2: stOut.stP51A_S1HandBs.bLedSelect02 := SEL(plant.fbSt020OvenB.State > eComponentState_running, TRUE, Statics.stPulse.bToggle1000ms);
	3: stOut.stP51A_S1HandBs.bLedSelect03 := SEL(plant.fbSt030Handling.State > eComponentState_running, TRUE, Statics.stPulse.bToggle1000ms);
	4: stOut.stP51A_S1HandBs.bLedSelect04 := SEL(plant.fbSt040Storage.State > eComponentState_running, TRUE, Statics.stPulse.bToggle1000ms);
	5: stOut.stP51A_S1HandBs.bLedSelect05 := SEL(plant.fbSt050Mould.State > eComponentState_running, TRUE, Statics.stPulse.bToggle1000ms);
	
END_CASE

stOut.stP51A_S1HandBs.bLedAlt := bAlternativ;

IF stIn.arrStStation[nSelStation].stManual.stManualAxis.eJogMode = E_Axis_JogMode.eJogMode_0 THEN
	stOut.stP51A_S1HandBs.bLedDistance := FALSE;
	stOut.stP51A_S1HandBs.bLedJog := TRUE;
ELSIF stIn.arrStStation[nSelStation].stManual.stManualAxis.eJogMode = E_Axis_JogMode.eJogMode_1 THEN
	stOut.stP51A_S1HandBs.bLedDistance := FALSE;
	stOut.stP51A_S1HandBs.bLedJog := FALSE;
ELSIF stIn.arrStStation[nSelStation].stManual.stManualAxis.eJogMode = E_Axis_JogMode.eJogMode_2 THEN
	stOut.stP51A_S1HandBs.bLedDistance := TRUE;
	stOut.stP51A_S1HandBs.bLedJog := FALSE;
END_IF
END_METHOD

METHOD PRIVATE M_PlcToHmi : BOOL
VAR
	bEn 	: BOOL;
	fVal	: LREAL;
END_VAR
/// general
//stOut.bLed_Reset := stOut.stCommon.stMain.stButton_Reset.bLed;
//stOut.bLed_Start := stOut.stCommon.stMain.stButton_Start.bLed;
//stOut.bLed_Tipp := stOut.stCommon.stMain.stButton_Step.bLed;
//stOut.bLed_GRST := stOut.stCommon.stMain.stButton_Home.bLed;
bLedTest := P_HMI_Controller.bLedTest;

// e.g. ..AND/OR... SafeArea1Ok...
stOut.stP50A_Haupt.bLedQuit := bLedTest OR stOut.stCommon.stSafety.bLedResetAreaST10;
//stOut.stP10A_Pult.bLedQuitLs := bLedTest;

/// specific

// +P10A/B/C Oven
//stOut.stP10A_Pult.bLedRichtungL/R := bLedTest OR stOut.stSt010.LedRichtungL/R;	// LedRichtungL/R; LDT-BU, 2FDI-NO, 1DO; P10A-51SJ3


// LED module / Ampel
(* IO.stControlCabinetIO.stOut.stA02.bLedModAllgRt :=  bLedTest OR (stPulse.bToggle500ms AND stGlobalModuleInfo.eHeaderPriority = E_AlarmPriority.Error);
IO.stControlCabinetIO.stOut.stA02.bLedModAllgGe :=  bLedTest OR (stPulse.bToggle500ms AND stGlobalModuleInfo.eHeaderPriority = E_AlarmPriority.Warning);
IO.stControlCabinetIO.stOut.stA02.bLedModAllgGn :=  bLedTest OR (stGlobalModuleInfo.eHeaderPriority <> E_AlarmPriority.Error AND 
															     stGlobalModuleInfo.eHeaderPriority <> E_AlarmPriority.Warning AND 
																 stGlobalModuleInfo.astModuleStationsInfo[E_Module.eModule_M001].bStation_All_Started);
																 
IO.stControlCabinetIO.stOut.stA02.bLedModAllgBl :=  bLedTest OR (stPulse.bToggle500ms AND (stSt010IOvenA.bEnde OR stSt010IOvenA.bFehlstelle)); *)
END_METHOD

/// reset
METHOD M_Reset : BOOL
VAR
END_VAR
M_Reset := SUPER^.M_Reset();

bRequestManualControl := FALSE;
bRequestRecipeMgmt := FALSE;
bRequestSettingMgmt := FALSE;
bRequestUserMgmt := FALSE;
END_METHOD

METHOD M_Run : BOOL
VAR
END_VAR
IF NOT SUPER^.M_Run() THEN
	RETURN;
END_IF

M_HmiToPlc();
M_EuchnerToPlc();

M_PlcToHmi();
M_PlcToEuchner();

M_Run := TRUE;
END_METHOD

METHOD M_SetReferences : BOOL
VAR_IN_OUT
	stRefIn		: HMI_PROVIDER_HW_IN;
	stRefOut	: HMI_PROVIDER_HW_OUT;	
END_VAR
M_SetReferences := SUPER^.M_SetReferencesBase(stRefIn, stRefOut);
stIn REF= stRefIn;
stOut REF= stRefOut;
END_METHOD

PROPERTY RefsValid : bool
GET
RefsValid := SUPER^.RefsValid AND_THEN
			 __ISVALIDREF (stOut) AND_THEN
			 __ISVALIDREF (stIn);
END_GET
END_PROPERTY

END_FUNCTION_BLOCK

// ---- POUs/HMI/Provider/_Base/FB_HMI_PROVIDER_BASE.TcPOU
FUNCTION_BLOCK PUBLIC ABSTRACT FB_HMI_PROVIDER_BASE IMPLEMENTS ITF_HMI_PROVIDER
VAR_INPUT
END_VAR
VAR_OUTPUT
END_VAR
VAR
	eProvider	: E_HMI_PROVIDER;
	
	stItfHmiIn	: REFERENCE TO ST_HMI_IN;
	stItfHmiOut	: REFERENCE TO ST_HMI_OUT;
	
	bRequestManualControl,
	bRequestRecipeMgmt,
	bRequestSettingMgmt,
	bRequestUserMgmt,
	bMute		: BOOL;
END_VAR

PROPERTY ItfHmiIn : REFERENCE TO ST_HMI_IN
GET
ItfHmiIn REF= stItfHmiIn;
END_GET
END_PROPERTY

PROPERTY ItfHmiOut : REFERENCE TO ST_HMI_OUT
GET
ItfHmiOut REF= stItfHmiOut;
END_GET
END_PROPERTY

METHOD PUBLIC M_Init : BOOL
VAR_INPUT
END_VAR
P_HMI_Controller.M_RegisterProvider(THIS^);
M_Init := TRUE;
END_METHOD

(* reset*)
METHOD M_Reset : BOOL
stItfHmiIn.stSpecial.stButton_LedTest.bClick := FALSE;
END_METHOD

METHOD M_Run : BOOL
VAR
	msg : STRING;
END_VAR
IF NOT RefsValid THEN
	msg := CONCAT('HMI provider ref error, provider: ', TO_STRING(eProvider));
	Services.fbEventHandler.Select(TC_Events.SystemEventClass.ErrorEvent).ArgSetString(msg).Raise();
	RETURN;
END_IF

M_Run := TRUE;
END_METHOD

METHOD M_SetReferencesBase : BOOL
VAR_IN_OUT
	stHmiPrvIn	: ST_HMI_IN;
	stHmiPrvOut	: ST_HMI_OUT;
END_VAR
stItfHmiIn REF= stHmiPrvIn;
stItfHmiOut REF= stHmiPrvOut;
stItfHmiOut.stCommon REF= HMI.stHmi.stOut.stCommon; // same common out 4 all HMI provider, in order to save memory
M_SetReferencesBase := TRUE;
END_METHOD

PROPERTY Mute : bool
GET
Mute := bMute;
END_GET
END_PROPERTY

{attribute 'monitoring' := 'call'}
PROPERTY Provider : E_HMI_PROVIDER
GET
Provider := eProvider;
END_GET
END_PROPERTY

{attribute 'monitoring' := 'call'}
PROPERTY RefsValid : bool
GET
RefsValid := __ISVALIDREF (stItfHmiIn) AND_THEN
			 __ISVALIDREF (stItfHmiOut);
END_GET
END_PROPERTY

(* HMI control request (Bedienhoheit)
	set ti true, on any control request from the HMI provider (e.g.: watch IN struct)
	reset will be done by HMI controller, on other provider request  *)
{attribute 'monitoring':='call'}
PROPERTY RequestManualControl : BOOL
GET
RequestManualControl := bRequestManualControl;
END_GET
SET
bRequestManualControl := RequestManualControl;
END_SET
END_PROPERTY

(* HMI recipe control request (Bedienhoheit)  *)
{attribute 'monitoring':='call'}
PROPERTY RequestRecipeMgmt : BOOL
GET
RequestRecipeMgmt := bRequestRecipeMgmt;
END_GET
SET
bRequestRecipeMgmt := RequestRecipeMgmt;
END_SET
END_PROPERTY

(* HMI recipe control request (Bedienhoheit)  *)
{attribute 'monitoring':='call'}
PROPERTY RequestSettingMgmt : BOOL
GET
RequestSettingMgmt := bRequestSettingMgmt;
END_GET
SET
bRequestSettingMgmt := RequestSettingMgmt;
END_SET
END_PROPERTY

(* HMI user management control request (Bedienhoheit)  *)
{attribute 'monitoring':='call'}
PROPERTY RequestUserMgmt : BOOL
GET
RequestUserMgmt := bRequestUserMgmt;
END_GET
SET
bRequestUserMgmt := RequestUserMgmt;
END_SET
END_PROPERTY

END_FUNCTION_BLOCK

// ---- POUs/HMI/Provider/Tc3Hmi/FB_HMI_Provider_TC3.TcPOU
FUNCTION_BLOCK FB_HMI_Provider_TC3 EXTENDS FB_HMI_PROVIDER_BASE
VAR_OUTPUT
END_VAR
VAR
	ILog	: I_Logger;
	stIn	: REFERENCE TO ST_FromTc3Hmi;
	stOut	: REFERENCE TO ST_ToTc3Hmi;

	fbCounter			: FB_CounterHandling;
	
	nPopupToken			: INT;
	bResetToken			: BOOL;
	tonResetToken		: TON;
	
	stInMain_Mirror		: ST_HMI_BASE_CONTROL_IN;
END_VAR

METHOD M_Counter : BOOL
VAR_INPUT
END_VAR
VAR
END_VAR

// counter handling
fbCounter(eUserLevel := HMI.eUserLevel, stControlCounterIn := stIn.stControlCounter, stControlCounterOut := stOut.stControlCounter, stCounter := HMI.stCounter, stCounterView := stOut.stCounter);
END_METHOD

METHOD PRIVATE M_HmiToPlc : BOOL
VAR
END_VAR

// map specific in
M_SpecificIn();
M_HmiToPlc := TRUE;
END_METHOD

METHOD PUBLIC M_Init : BOOL
VAR_INPUT
END_VAR
VAR
	ii		: INT;
END_VAR
//aSClearText[EN] := 'Initialize TC3 HMI';

// set up defaults
eProvider := E_HMI_PROVIDER.eHmiProvider_TC3HMI;
ILog := SERVICES.ILog;
M_SetReferences(HMI.stHmiTc3.stOut, HMI.stHmiTc3.stIn);

// recipe, settings and user management done only by this provider
bRequestRecipeMgmt := TRUE;
bRequestSettingMgmt := TRUE;
bRequestUserMgmt := TRUE;

FOR ii := 0 TO 30 DO
	stOut.stSetupPlant[ii].stGet.wsName := stOut.stSetupPlant[ii].stGet.wsNameId := "0";
	stOut.stSetupPlant[ii].stSet.wsName := stOut.stSetupPlant[ii].stSet.wsNameId := "0";
	stOut.stSetupPlant[ii].stState.wsName := stOut.stSetupPlant[ii].stState.wsNameId := "0";
END_FOR

M_SpecificInit();

//aSClearText[EN] := 'HMI init done.';
M_Init := SUPER^.M_Init();
END_METHOD

METHOD PRIVATE M_PlcToHmi : BOOL
VAR
	ii, nn, nnn	: DINT;
END_VAR
// map HMI provider interface out to TC3 hmi (mapping of common out not needed anymore, due to reference type!)
//stTc3HmiOut.stCommon := stItfHmiOut.stCommon;

//---------------------------------------------------------------------------------------------------------------------------------------------
// system time and date
stOut.stHeader.sDateAndTime := LEFT (Statics.sTimeString, 19);

//language
stOut.stHeader.nLanguageList := 2;
stOut.stHeader.aLanguageList[0] := CONST.stTextListGlobal.stText_EN;
stOut.stHeader.aLanguageList[1] := CONST.stTextListGlobal.stText_DE;
stOut.stHeader.aLanguageList[2] := CONST.stTextListGlobal.stText_BE;

stOut.stHeader.stMessageBox1 := CONST.stTextListGlobal.stText_AllOk;
stOut.stHeader.stMessageBox2 := CONST.stTextListGlobal.stText_notextempty;
stOut.stHeader.stMessageBox3 := CONST.stTextListGlobal.stText_notextempty;

stOut.stHeader.stMessageBox1Color.color := F_ColorToStringHexColor(STATICS.stColor.Theme);
stOut.stHeader.stMessageBox2Color.color := F_ColorToStringHexColor(STATICS.stColor.Theme);
stOut.stHeader.stMessageBox3Color.color := F_ColorToStringHexColor(STATICS.stColor.Theme);

//---------------------------------------------------------------------------------------------------------------------------------------------
// default buttons

//set button language
stOut.stControlCounter.stButtonSave.stName := stTextListGlobal.stText_Save;

//--------------------------------------------------------------------------------------------------------------
// safety - ES
// safety - ES dynamic (loop)
//stOut.stEmergencyStop[0].nState := SEL(P_Safety.arrEmergencyStopState[E_EmergencyStop.eEmergencyStop_A1], 0, 1);
//stOut.stEmergencyStop[1].nState := SEL(P_Safety.arrEmergencyStopState[E_EmergencyStop.eEmergencyStop_M1P1], 0, 1);
//stOut.stEmergencyStop[2].nState := SEL(P_Safety.arrEmergencyStopState[E_EmergencyStop.eEmergencyStop_M1P2], 0, 1);

// doors
//stOut.stDoor[0].stStateColor.color := F_ColorToStringHexColor(P_Safety.fbDoor[1].iDoorStateCol);

M_SpecificOut();
M_PlcToHmi := TRUE;
END_METHOD

METHOD PRIVATE M_Popup : BOOL
VAR_INPUT
END_VAR
tonResetToken.IN := bResetToken;
tonResetToken.PT := T#1S;
tonResetToken();
IF tonResetToken.Q THEN
	bResetToken := FALSE;
	M_PopupReset();
END_IF
END_METHOD

METHOD PUBLIC M_PopupCheck : BOOL
VAR_INPUT
	nToken		: INT;
END_VAR
M_PopupCheck := (nPopupToken = 0) or (nPopupToken = nToken);
END_METHOD

METHOD PUBLIC M_PopupReset : BOOL
VAR_INPUT
END_VAR
nPopupToken := 0;
stOut.stPopup.bVisible := FALSE;
END_METHOD

METHOD PUBLIC M_PopupSet : INT
VAR_INPUT
	nToken			: int;
	stText			: ST_TEXT;
	stNameButton01	: ST_Text;
	stNameButton02	: ST_Text;
	stNameButton03	: ST_Text;
	stNameButton04	: ST_Text;
END_VAR
M_PopupSet := 0;
nPopupToken := nToken;
stOut.stPopup.bVisible := TRUE;
stOut.stPopup.stText := stText;
stOut.stPopup.bButton01:= FALSE;
stOut.stPopup.bButton02:= FALSE;
stOut.stPopup.bButton03:= FALSE;
stOut.stPopup.bButton04:= FALSE;
IF stNameButton01.wsNameId <>"" THEN
	stOut.stPopup.bButton01:= TRUE;
	stOut.stPopup.stButton01.stName := stNameButton01;
END_IF
IF stNameButton02.wsNameId <>"" THEN
	stOut.stPopup.bButton02:= TRUE;
	stOut.stPopup.stButton02.stName := stNameButton02;
END_IF
IF stNameButton03.wsNameId <>"" THEN
	stOut.stPopup.bButton03:= TRUE;
	stOut.stPopup.stButton03.stName := stNameButton03;
END_IF
IF stNameButton04.wsNameId <>"" THEN
	stOut.stPopup.bButton04:= TRUE;
	stOut.stPopup.stButton04.stName := stNameButton04;
END_IF
IF  HMI.stHmiTc3.stIn.stPopup.stButton01.bClick THEN
	bResetToken	:= true;
	M_PopupSet := 1;
ELSIF HMI.stHmiTc3.stIn.stPopup.stButton02.bClick THEN
	bResetToken	:= TRUE;
	M_PopupSet := 2;	
ELSIF HMI.stHmiTc3.stIn.stPopup.stButton03.bClick THEN
	bResetToken	:= TRUE;
	M_PopupSet := 3;	
ELSIF HMI.stHmiTc3.stIn.stPopup.stButton04.bClick THEN
	bResetToken	:= TRUE;
	M_PopupSet := 4;		
END_IF
IF M_PopupSet <> 0 THEN
	stOut.stPopup.bVisible := FALSE;
END_IF
END_METHOD

/// reset
METHOD M_Reset : BOOL
VAR
END_VAR
M_Reset := SUPER^.M_Reset();

M_PopupReset();

bRequestManualControl := FALSE;
// recipe, settings and user management done only by this provider
//bRequestRecipeMgmt := FALSE;
//bRequestSettingMgmt := FALSE;
//bRequestUserMgmt := FALSE;
END_METHOD

METHOD M_Run : BOOL
VAR_INST
	tofCleanScreen		: TOF;
	arrModuleManMir	: ARRAY[0..E_Module.eModule_nMaxIdx] OF ST_HMI_BASE_MODULE_MANUAL_IN;
	arrStationManMir	: ARRAY[0..E_Station.eStation_nMaxIdx] OF ST_HMI_BASE_STATION_MANUAL_IN;
END_VAR
VAR
	ii : INT;
END_VAR
IF NOT SUPER^.M_Run() THEN
	RETURN;
END_IF

// chk control request, e.g.: watch for changes --> stIn.arrStStation[xx].stManual...
// modules
FOR ii := 0 TO E_Module.eModule_nMaxIdx DO
	IF P_Plant.aIModule[ii] = 0 THEN CONTINUE; END_IF
	
	IF (MEMCMP(ADR(arrModuleManMir[ii]), ADR(stIn.arrStModule[ii].stManual), SIZEOF(arrModuleManMir[ii])) <> 0) THEN
		bRequestManualControl := TRUE; // request manual control on any change in .stManual. ...
	END_IF
	MEMCPY(ADR(arrModuleManMir[ii]), ADR(stIn.arrStModule[ii].stManual), SIZEOF(arrModuleManMir[ii]));
END_FOR
FOR ii := 0 TO E_Station.eStation_nMaxIdx DO	
	IF P_Plant.aIStaton[ii] = 0 THEN CONTINUE; END_IF
	
	IF (MEMCMP(ADR(arrStationManMir[ii]), ADR(stIn.arrStStation[ii].stManual), SIZEOF(arrStationManMir[ii])) <> 0) THEN
		bRequestManualControl := TRUE; // request manual control on any change in .stManual. ...
	END_IF
	MEMCPY(ADR(arrStationManMir[ii]), ADR(stIn.arrStStation[ii].stManual), SIZEOF(arrStationManMir[ii]));
END_FOR

// recipe, settings and user management done only by this provider
bRequestRecipeMgmt := TRUE;
bRequestSettingMgmt := TRUE;
bRequestUserMgmt := TRUE;

tofCleanScreen(IN := stHmi.stIn.stSpecial.stButton_CleanScreen.bClick, PT := T#1M, Q => bMute);

M_HmiToPlc(); 
M_Counter();
M_PlcToHmi();

M_Run := TRUE;
END_METHOD

METHOD M_SetReferences : BOOL
VAR_IN_OUT
	stToTc3Hmi		: ST_ToTc3Hmi;
	stFromTc3Hmi	: ST_FromTc3Hmi;
END_VAR
M_SetReferences := SUPER^.M_SetReferencesBase(stFromTc3Hmi, stToTc3Hmi);
stOut REF= stToTc3Hmi;
stIn REF= stFromTc3Hmi;
END_METHOD

METHOD INTERNAL M_SpecificIn : BOOL
VAR_INPUT
END_VAR
VAR
END_VAR
// stations
END_METHOD

METHOD INTERNAL M_SpecificInit : BOOL
VAR_INPUT
END_VAR
VAR
	nn : INT;
END_VAR
// init project specific HMI provider stuff here

(* stTc3HmiOut.stSetupPlant[1].stStation := stTextListGlobal.stText_ST005_NameId;
stTc3HmiOut.stSetupPlant[1].stName := stTextListGlobal.stText_Drehwerkzeug;
stTc3HmiOut.stSetupPlant[2].stStation := stTextListGlobal.stText_ST005_NameId;
stTc3HmiOut.stSetupPlant[2].stName := stTextListGlobal.stText_Kontaktwerkzeug1;
stTc3HmiOut.stSetupPlant[3].stStation := stTextListGlobal.stText_ST005_NameId;
stTc3HmiOut.stSetupPlant[3].stName := stTextListGlobal.stText_Kontaktwerkzeug2; *)


nn:=1;
stOut.stEmergencyStop[nn].stName := stTextListGlobal.stText_Emergencystop_A1P1;
stOut.stEmergencyStop[nn].stItem.wsName := stOut.stEmergencyStop[nn].stItem.wsNameId := "++A1+P1-6S2";
nn:=nn+1;
stOut.stEmergencyStop[nn].stName := stTextListGlobal.stText_Emergencystop_M1P1;
stOut.stEmergencyStop[nn].stItem.wsName := stOut.stEmergencyStop[nn].stItem.wsNameId := "++M1+P1-2S1";
nn:=nn+1;
stOut.stEmergencyStop[nn].stName := stTextListGlobal.stText_Emergencystop_M1P2;
stOut.stEmergencyStop[nn].stItem.wsName := stOut.stEmergencyStop[nn].stItem.wsNameId := "++M1+P2-2S1";


nn:=1;
stOut.stDoor[nn].stName := stTextListGlobal.stText_Modul1_Schott1;
stOut.stDoor[nn].stItem.wsName := stOut.stDoor[nn].stItem.wsNameId := "++M1+PSEN_001-2S2";
nn:=nn+1;
stOut.stDoor[nn].stName := stTextListGlobal.stText_Modul1_Door1;
stOut.stDoor[nn].stItem.wsName := stOut.stDoor[nn].stItem.wsNameId := "++M1+PSEN_002-2S2";
nn:=nn+1;
stOut.stDoor[nn].stName := stTextListGlobal.stText_Modul1_Door2;
stOut.stDoor[nn].stItem.wsName := stOut.stDoor[nn].stItem.wsNameId := "++M1+PSEN_003-2S2";
nn:=nn+1;
stOut.stDoor[nn].stName := stTextListGlobal.stText_Modul1_Door3;
stOut.stDoor[nn].stItem.wsName := stOut.stDoor[nn].stItem.wsNameId := "++M1+PSEN_004-2S2";
nn:=nn+1;
stOut.stDoor[nn].stName := stTextListGlobal.stText_Modul1_Door4;
stOut.stDoor[nn].stItem.wsName := stOut.stDoor[nn].stItem.wsNameId := "++M1+PSEN_005-2S2";
nn:=nn+1;
stOut.stDoor[nn].stName := stTextListGlobal.stText_Modul1_Schott2;
stOut.stDoor[nn].stItem.wsName := stOut.stDoor[nn].stItem.wsNameId := "++M1+E2-73BG7";

// stations, e.g.:
//stTc3HmiOut.astStation[E_Station.eStation_ST010_OvenA].astButton[1] := stItfHmiOut.stSt010.stButtonOvenAxx1;
//stTc3HmiOut.astStation[E_Station.eStation_ST010_OvenA].stEingabeStatusColor := stItfHmiOut.stSt010.stOvenAStatusColor;
//stTc3HmiOut.astStation[E_Station.eStation_ST010_OvenA].stEingabeStatus := stItfHmiOut.stSt010.stOvenAStatus;
//stTc3HmiOut.astStation[E_Station.eStation_ST010_OvenA].astButton[2] := stItfHmiOut.stSt010.stButtonOvenAxx2;


//aSClearText[EN] := 'HMI init done.';
M_SpecificInit := TRUE;
END_METHOD

METHOD INTERNAL M_SpecificOut : BOOL
VAR_INPUT
END_VAR
VAR
END_VAR
//stOut.stConditionMonitoring.fVoltage_L1 := IO.stControlCabinetIO.stIn.stDevice_MonitoringVoltage400Vac.fL1_Voltage;
//stOut.stConditionMonitoring.fVoltage_L2 := IO.stControlCabinetIO.stIn.stDevice_MonitoringVoltage400Vac.fL2_Voltage;
//stOut.stConditionMonitoring.fVoltage_L3 := IO.stControlCabinetIO.stIn.stDevice_MonitoringVoltage400Vac.fL3_Voltage;
//stOut.stConditionMonitoring.fVoltage_L1_L2 := IO.stControlCabinetIO.stIn.stDevice_MonitoringVoltage400Vac.fL1_L2Voltage;
//stOut.stConditionMonitoring.fVoltage_L2_L3 := IO.stControlCabinetIO.stIn.stDevice_MonitoringVoltage400Vac.fL2_L3Voltage;
//stOut.stConditionMonitoring.fVoltage_L3_L1 := IO.stControlCabinetIO.stIn.stDevice_MonitoringVoltage400Vac.fL3_L1Voltage;
//stOut.stConditionMonitoring.fPowerFactor := IO.stControlCabinetIO.stIn.stDevice_MonitoringVoltage400Vac.fPowerQualityFactor;
stOut.stConditionMonitoring.fCurrent_L1 := 0;
stOut.stConditionMonitoring.fCurrent_L2 := 0;
stOut.stConditionMonitoring.fCurrent_L3 := 0;

// stations
//stTc3HmiOut.astStation[E_Station.eStation_ST010_OvenA].astButton[1] := stItfHmiOut.stSt010.stButtonOvenAxx1;
//stTc3HmiOut.astStation[E_Station.eStation_ST010_OvenA].stEingabeStatusColor := stItfHmiOut.stSt010.stOvenAStatusColor;
//stTc3HmiOut.astStation[E_Station.eStation_ST010_OvenA].stEingabeStatus := stItfHmiOut.stSt010.stOvenAStatus;
//stTc3HmiOut.astStation[E_Station.eStation_ST010_OvenA].astButton[2] := stItfHmiOut.stSt010.stButtonOvenAxx2;
END_METHOD

PROPERTY RefsValid : bool
GET
RefsValid := SUPER^.RefsValid AND_THEN
			 __ISVALIDREF (stOut) AND_THEN
			 __ISVALIDREF (stIn);
END_GET
END_PROPERTY

END_FUNCTION_BLOCK

// ---- POUs/HMI/Utilities/FB_CounterHandling.TcPOU
FUNCTION_BLOCK FB_CounterHandling
VAR_INPUT
	eUserLevel			: E_User_Level;
END_VAR
VAR_IN_OUT
	stControlCounterIn	: ST_CounterControlIn;
	stControlCounterOut	: ST_CounterControlOut;
	stCounter			: ARRAY[0..CONST.iMaxIdxCounter] OF ST_Counter_Item;
	stCounterView		: ARRAY[0..CONST.iMaxIdxCounter] OF ST_Counter_Item_String;
END_VAR
VAR_OUTPUT
	stInfo					: ST_Text;
	eSupervisionReaction	: E_CounterReaction;
	stSupervison			: ST_Text;
END_VAR
VAR
	ii				: DINT;
	bInit			: BOOL;
	rtSave			: R_TRIG;
	rtReset			: R_TRIG;
	nColumnIndex	: INT;
	nRowIndex		: INT;
	tofInfo			: TOF;
END_VAR


nColumnIndex	:= stControlCounterIn.nSelectedColumIndex + 1;
nRowIndex		:= stControlCounterIn.nSelectedRowIndex + 1;

IF NOT bInit THEN
	bInit:= TRUE;
	stControlCounterOut.stButtonSave.stName := F_CreateDynText("save",0);
	stControlCounterOut.stButtonReset.stName := F_CreateDynText("reset",0);
END_IF

stControlCounterOut.stButtonSave.stColor.color := SEL(stControlCounterIn.stButtonSave.bClick, 
													F_ColorToStringHexColor(STATICS.stColor.Theme),
													F_ColorToStringHexColor(STATICS.stColor.LimeGreen));

stControlCounterOut.stButtonReset.stColor.color := SEL(stControlCounterIn.stButtonReset.bClick,
													F_ColorToStringHexColor(STATICS.stColor.Theme),
													F_ColorToStringHexColor(STATICS.stColor.LimeGreen));

stControlCounterOut.bVisible_Number := FALSE;
stControlCounterOut.bVisible_String := FALSE;
stControlCounterOut.bVisible_UserLevel := FALSE;
stControlCounterOut.bVisible_Reaction := FALSE;

stControlCounterOut.nUserLevelUsers := (E_User_Level.eUser_Level_nMaxIdx);
stControlCounterOut.aUserLevelUsers[0] := CONST.stTextListGlobal.stText_UserLevel00;
stControlCounterOut.aUserLevelUsers[1] := CONST.stTextListGlobal.stText_UserLevel01;
stControlCounterOut.aUserLevelUsers[2] := CONST.stTextListGlobal.stText_UserLevel02;
stControlCounterOut.aUserLevelUsers[3] := CONST.stTextListGlobal.stText_UserLevel03;
stControlCounterOut.aUserLevelUsers[4] := CONST.stTextListGlobal.stText_UserLevel04;
stControlCounterOut.aUserLevelUsers[5] := CONST.stTextListGlobal.stText_UserLevel05;
stControlCounterOut.aUserLevelUsers[6] := CONST.stTextListGlobal.stText_UserLevel06;

stControlCounterOut.nReaction := E_EventReaction.Undefined;
stControlCounterOut.aReaction[0] := CONST.stTextListGlobal.stText_Counter_Reaction_None;
stControlCounterOut.aReaction[1] := CONST.stTextListGlobal.stText_Counter_Reaction_Info;
stControlCounterOut.aReaction[2] := CONST.stTextListGlobal.stText_Counter_Reaction_Warning;
stControlCounterOut.aReaction[3] := CONST.stTextListGlobal.stText_Counter_Reaction_Error;
stControlCounterOut.aReaction[4] := CONST.stTextListGlobal.stText_Counter_Reaction_SerialError_Warning;
stControlCounterOut.aReaction[5] := CONST.stTextListGlobal.stText_Counter_Reaction_SerialError_Warning_Stop;

rtSave(CLK := stControlCounterIn.stButtonSave.bClick);
rtReset(CLK := stControlCounterIn.stButtonReset.bClick);

//clear settins view
MEMSET(ADR(stCounterView), 0, SIZEOF(stCounterView));
FOR ii := 0 TO CONST.iMaxIdxCounter DO
	M_SetUpCounterViewTxt(stCounter[ii], stCounterView[ii]);
	M_SetUpCounterReaction(stCounter[ii]);
	M_SetUpCounterState(stCounter[ii]);	
END_FOR

//monitoring for control
CASE nColumnIndex OF

	1: // rfid
		//IF (stSettings[nRowIndex].eDataType <> E_DataType.eDataType_None) THEN
		//	
		//END_IF
		;	
	5,7,9,11,13,15:	// id
		stControlCounterOut.bVisible_Number := TRUE;	

	6,8:// id
		stControlCounterOut.bVisible_Reaction := TRUE;
		stControlCounterOut.nReaction := (E_CounterReaction.eCounterReaction_Max -2);	
		
	10,12:// id
		stControlCounterOut.bVisible_Reaction := TRUE;
		stControlCounterOut.nReaction := (E_CounterReaction.eCounterReaction_Max);

	14,16:// id
		stControlCounterOut.bVisible_Reaction := TRUE;		
		stControlCounterOut.nReaction := (E_CounterReaction.eCounterReaction_Max -2);
		
	17: // unit user level programmer
		IF (eUserLevel < E_User_Level.eUser_Level_Programmer) THEN
			tofInfo.IN :=	TRUE;
			stInfo.wsName := "incorrect user level";
			stInfo.wsNameId := "incorrectuserlevel";
		ELSE
			stControlCounterOut.bVisible_UserLevel := TRUE;	
		END_IF			
		
END_CASE

IF rtReset.Q THEN
	IF (eUserLevel < stCounter[nRowIndex].eUserLevel) THEN
		tofInfo.IN :=	TRUE;
		stInfo.wsName := "incorrect user level";
		stInfo.wsNameId := "incorrectuserlevel";					
	ELSE	
		stCounter[nRowIndex].nValueOk := 0;
		stCounter[nRowIndex].nValueNok := 0;
		tofInfo.IN :=	TRUE;
		stInfo.wsName := "Zähler rückgesetzt";
		stInfo.wsNameId := "counterreseted";	
	END_IF
END_IF	
	

IF rtSave.Q THEN
	IF (eUserLevel < stCounter[nRowIndex].eUserLevel) THEN
		tofInfo.IN :=	TRUE;
		stInfo.wsName := "incorrect user level";
		stInfo.wsNameId := "incorrectuserlevel";					
	ELSE	
		CASE nColumnIndex OF
		
			1: // name only write by programmer
				IF (eUserLevel < E_User_Level.eUser_Level_Manager) THEN
					tofInfo.IN :=	TRUE;
					stInfo.wsName := "incorrect user level";
					stInfo.wsNameId := "incorrectuserlevel";
				ELSE
					stCounter[nRowIndex].stGroup.wsName := stCounter[nRowIndex].stGroup.wsNameId := stControlCounterIn.wsInputString;
				END_IF
			2,3,4: // name only write by program
				;

			5: // Level
				IF (eUserLevel < stCounter[nRowIndex].eUserLevel) THEN
					tofInfo.IN :=	TRUE;
					stInfo.wsName := "incorrect user level";
					stInfo.wsNameId := "incorrectuserlevel";
				ELSE
					stCounter[nRowIndex].nValueOkLevel1 := stControlCounterIn.nInputNumber;
				END_IF 

			6: // Reaction
				IF (eUserLevel < stCounter[nRowIndex].eUserLevel) THEN
					tofInfo.IN :=	TRUE;
					stInfo.wsName := "incorrect user level";
					stInfo.wsNameId := "incorrectuserlevel";
				ELSE
					stCounter[nRowIndex].eReactionOkLevel1 := stControlCounterIn.eReaction;
				END_IF

			7: // Level
				IF (eUserLevel < stCounter[nRowIndex].eUserLevel) THEN
					tofInfo.IN :=	TRUE;
					stInfo.wsName := "incorrect user level";
					stInfo.wsNameId := "incorrectuserlevel";
				ELSE
					stCounter[nRowIndex].nValueOkLevel2 := stControlCounterIn.nInputNumber;
				END_IF				

			8: // Reaction
				IF (eUserLevel < stCounter[nRowIndex].eUserLevel) THEN
					tofInfo.IN :=	TRUE;
					stInfo.wsName := "incorrect user level";
					stInfo.wsNameId := "incorrectuserlevel";
				ELSE
					stCounter[nRowIndex].eReactionOkLevel2 := stControlCounterIn.eReaction;
				END_IF
				
			9: // Level
				IF (eUserLevel < stCounter[nRowIndex].eUserLevel) THEN
					tofInfo.IN :=	TRUE;
					stInfo.wsName := "incorrect user level";
					stInfo.wsNameId := "incorrectuserlevel";
				ELSE
					stCounter[nRowIndex].nValueNokLevel1 := stControlCounterIn.nInputNumber;
				END_IF	

			10: // Reaction
				IF (eUserLevel < stCounter[nRowIndex].eUserLevel) THEN
					tofInfo.IN :=	TRUE;
					stInfo.wsName := "incorrect user level";
					stInfo.wsNameId := "incorrectuserlevel";
				ELSE
					stCounter[nRowIndex].eReactionNokLevel1 := stControlCounterIn.eReaction;
				END_IF				
				
			11: // Level
				IF (eUserLevel < stCounter[nRowIndex].eUserLevel) THEN
					tofInfo.IN :=	TRUE;
					stInfo.wsName := "incorrect user level";
					stInfo.wsNameId := "incorrectuserlevel";
				ELSE
					stCounter[nRowIndex].nValueNokLevel2 := stControlCounterIn.nInputNumber;
				END_IF

			12: // Reaction
				IF (eUserLevel < stCounter[nRowIndex].eUserLevel) THEN
					tofInfo.IN :=	TRUE;
					stInfo.wsName := "incorrect user level";
					stInfo.wsNameId := "incorrectuserlevel";
				ELSE
					stCounter[nRowIndex].eReactionNokLevel2 := stControlCounterIn.eReaction;
				END_IF				
				
			13: // Level
				IF (eUserLevel < stCounter[nRowIndex].eUserLevel) THEN
					tofInfo.IN :=	TRUE;
					stInfo.wsName := "incorrect user level";
					stInfo.wsNameId := "incorrectuserlevel";
				ELSE
					stCounter[nRowIndex].nValueTotalLevel1 := stControlCounterIn.nInputNumber;
				END_IF

			14: // Reaction
				IF (eUserLevel < stCounter[nRowIndex].eUserLevel) THEN
					tofInfo.IN :=	TRUE;
					stInfo.wsName := "incorrect user level";
					stInfo.wsNameId := "incorrectuserlevel";
				ELSE
					stCounter[nRowIndex].eReactionTotalLevel1 := stControlCounterIn.eReaction;
				END_IF
				
			15: // Level
				IF (eUserLevel < stCounter[nRowIndex].eUserLevel) THEN
					tofInfo.IN :=	TRUE;
					stInfo.wsName := "incorrect user level";
					stInfo.wsNameId := "incorrectuserlevel";
				ELSE
					stCounter[nRowIndex].nValueTotalLevel2 := stControlCounterIn.nInputNumber;
				END_IF			

			16: // Reaction
				IF (eUserLevel < stCounter[nRowIndex].eUserLevel) THEN
					tofInfo.IN :=	TRUE;
					stInfo.wsName := "incorrect user level";
					stInfo.wsNameId := "incorrectuserlevel";
				ELSE
					stCounter[nRowIndex].eReactionTotalLevel2 := stControlCounterIn.eReaction;
				END_IF				

			17: // recipe level manager
				IF (eUserLevel < E_User_Level.eUser_Level_Manager) 
					OR (stCounter[nRowIndex].eUserLevel = E_User_Level.eUser_Level_Programmer AND (eUserLevel <> E_User_Level.eUser_Level_Programmer))
				THEN
					tofInfo.IN :=	TRUE;
					stInfo.wsName := "incorrect user level";
					stInfo.wsNameId := "incorrectuserlevel";
				ELSE
					stCounter[nRowIndex].eUserLevel := stControlCounterIn.eUserLevel;
				END_IF 				
		END_CASE
	END_IF
END_IF

stSupervison := M_Supervision();

tofInfo(PT := T#2S, Q => stControlCounterOut.bVisibleInfo);
tofInfo.IN := FALSE;
stControlCounterOut.stInfo := stInfo;

METHOD PRIVATE M_SetUpCounterReaction : BOOL
VAR_IN_OUT
	stCnt	: ST_Counter_Item;
END_VAR
stCnt.eCurrentReactionOkLevel1 := 		E_CounterReaction.eCounterReaction_None;
stCnt.eCurrentReactionOkLevel2 := 		E_CounterReaction.eCounterReaction_None;
stCnt.eCurrentReactionNokLevel1 := 		E_CounterReaction.eCounterReaction_None;
stCnt.eCurrentReactionNokLevel2 := 		E_CounterReaction.eCounterReaction_None;
stCnt.eCurrentReactionTotalLevel1 := 	E_CounterReaction.eCounterReaction_None;
stCnt.eCurrentReactionTotalLevel2 := 	E_CounterReaction.eCounterReaction_None;

CASE stCnt.eReactionOkLevel1 OF 
	E_CounterReaction.eCounterReaction_SerialFault_Warning,
	E_CounterReaction.eCounterReaction_SerialFault_Error:
	stCnt.eCurrentReactionOkLevel1 :=	E_CounterReaction.eCounterReaction_None;
ELSE
	IF (stCnt.nValueOk >= stCnt.nValueOkLevel1) THEN
		stCnt.eCurrentReactionOkLevel1 := stCnt.eReactionOkLevel1;
	END_IF
END_CASE
CASE stCnt.eReactionOkLevel2 OF 
	E_CounterReaction.eCounterReaction_SerialFault_Warning,
	E_CounterReaction.eCounterReaction_SerialFault_Error:
	stCnt.eCurrentReactionOkLevel2 :=	E_CounterReaction.eCounterReaction_None;
ELSE
	IF (stCnt.nValueOk >= stCnt.nValueOkLevel2) THEN
		stCnt.eCurrentReactionOkLevel2 := stCnt.eReactionOkLevel2;
	END_IF
END_CASE


CASE stCnt.eReactionNokLevel1 OF 
	E_CounterReaction.eCounterReaction_SerialFault_Warning, 
	E_CounterReaction.eCounterReaction_SerialFault_Error:
	IF (stCnt.nValueSerialError >= stCnt.nValueNokLevel1) THEN
		stCnt.eCurrentReactionNokLevel1 := stCnt.eReactionNokLevel1;
	END_IF
ELSE
	IF (stCnt.nValueNok >= stCnt.nValueNokLevel1) THEN
		stCnt.eCurrentReactionNokLevel1 := stCnt.eReactionNokLevel1;
	END_IF
END_CASE
CASE stCnt.eReactionNokLevel2 OF 
	E_CounterReaction.eCounterReaction_SerialFault_Warning, 
	E_CounterReaction.eCounterReaction_SerialFault_Error:
	IF (stCnt.nValueSerialError >= stCnt.nValueNokLevel2) THEN
		stCnt.eCurrentReactionNokLevel2 := stCnt.eReactionNokLevel2;
	END_IF
ELSE
	IF (stCnt.nValueNok >= stCnt.nValueNokLevel2) THEN
		stCnt.eCurrentReactionNokLevel2 := stCnt.eReactionNokLevel2;
	END_IF	
END_CASE

IF (stCnt.nValueTotal >= stCnt.nValueTotalLevel1) THEN
	stCnt.eCurrentReactionTotalLevel1 := stCnt.eReactionTotalLevel1;
END_IF
IF (stCnt.nValueTotal >= stCnt.nValueTotalLevel2) THEN
	stCnt.eCurrentReactionTotalLevel2 := stCnt.eReactionTotalLevel2;
END_IF

M_setUpCounterReaction := TRUE;
END_METHOD

METHOD PRIVATE M_SetUpCounterState : BOOL
VAR_IN_OUT
	stCnt	: ST_Counter_Item;
END_VAR
//Counter State
stCnt.eCurrentCounterState := E_CounterReaction.eCounterReaction_None;
IF  stCnt.eCurrentReactionNokLevel1 = E_CounterReaction.eCounterReaction_SerialFault_Error THEN
	stCnt.eCurrentCounterState := E_CounterReaction.eCounterReaction_SerialFault_Error;
ELSIF stCnt.eCurrentReactionNokLevel2 = E_CounterReaction.eCounterReaction_SerialFault_Error THEN
	stCnt.eCurrentCounterState := E_CounterReaction.eCounterReaction_SerialFault_Error;
ELSIF stCnt.eCurrentReactionOkLevel1 = E_CounterReaction.eCounterReaction_Error THEN
	stCnt.eCurrentCounterState := E_CounterReaction.eCounterReaction_Error;
ELSIF stCnt.eCurrentReactionOkLevel2 = E_CounterReaction.eCounterReaction_Error THEN
	stCnt.eCurrentCounterState := E_CounterReaction.eCounterReaction_Error;
ELSIF stCnt.eCurrentReactionTotalLevel1 = E_CounterReaction.eCounterReaction_Error THEN
	stCnt.eCurrentCounterState := E_CounterReaction.eCounterReaction_Error;
ELSIF stCnt.eCurrentReactionTotalLevel2 = E_CounterReaction.eCounterReaction_Error THEN
	stCnt.eCurrentCounterState := E_CounterReaction.eCounterReaction_Error;	

ELSIF  stCnt.eCurrentReactionNokLevel1 = E_CounterReaction.eCounterReaction_SerialFault_Warning THEN
	stCnt.eCurrentCounterState := E_CounterReaction.eCounterReaction_SerialFault_Warning;
ELSIF stCnt.eCurrentReactionNokLevel2 = E_CounterReaction.eCounterReaction_SerialFault_Warning THEN
	stCnt.eCurrentCounterState := E_CounterReaction.eCounterReaction_SerialFault_Warning;
ELSIF stCnt.eCurrentReactionOkLevel1 = E_CounterReaction.eCounterReaction_Warning THEN
	stCnt.eCurrentCounterState := E_CounterReaction.eCounterReaction_Warning;
ELSIF stCnt.eCurrentReactionOkLevel2 = E_CounterReaction.eCounterReaction_Warning THEN
	stCnt.eCurrentCounterState := E_CounterReaction.eCounterReaction_Warning;
ELSIF stCnt.eCurrentReactionTotalLevel1 = E_CounterReaction.eCounterReaction_Warning THEN
	stCnt.eCurrentCounterState := E_CounterReaction.eCounterReaction_Warning;	
ELSIF stCnt.eCurrentReactionTotalLevel2 = E_CounterReaction.eCounterReaction_Warning THEN
	stCnt.eCurrentCounterState := E_CounterReaction.eCounterReaction_Warning;

ELSIF  stCnt.eCurrentReactionNokLevel1 = E_CounterReaction.eCounterReaction_Info THEN
	stCnt.eCurrentCounterState := E_CounterReaction.eCounterReaction_Info;
ELSIF stCnt.eCurrentReactionNokLevel2 = E_CounterReaction.eCounterReaction_Info THEN
	stCnt.eCurrentCounterState := E_CounterReaction.eCounterReaction_Info;
ELSIF stCnt.eCurrentReactionOkLevel1 = E_CounterReaction.eCounterReaction_Info THEN
	stCnt.eCurrentCounterState := E_CounterReaction.eCounterReaction_Info;
ELSIF stCnt.eCurrentReactionOkLevel2 = E_CounterReaction.eCounterReaction_Info THEN
	stCnt.eCurrentCounterState := E_CounterReaction.eCounterReaction_Info;
ELSIF stCnt.eCurrentReactionTotalLevel1 = E_CounterReaction.eCounterReaction_Info THEN
	stCnt.eCurrentCounterState := E_CounterReaction.eCounterReaction_Info;	
ELSIF stCnt.eCurrentReactionTotalLevel2 = E_CounterReaction.eCounterReaction_Info THEN
	stCnt.eCurrentCounterState := E_CounterReaction.eCounterReaction_Info;
ELSE
	stCnt.eCurrentCounterState := E_CounterReaction.eCounterReaction_None;
END_IF

M_SetUpCounterState := TRUE;
END_METHOD

METHOD PRIVATE M_SetUpCounterViewTxt : BOOL
VAR_IN_OUT
	stCnt	: ST_Counter_Item;
	stCntVw	: ST_Counter_Item_String;
END_VAR
IF (stCnt.stName.wsName = "") AND (stCnt.stName.wsNameId = "")  THEN
	stCntVw.stDataType.wsName := "";		
ELSIF stCnt.eDataType = E_DataType.eDataType_None THEN
	stCntVw.stDataType.wsName := stCntVw.stDataType.wsNameId :="none";	
ELSIF stCnt.eDataType = E_DataType.eDataType_bool THEN
	stCntVw.stDataType.wsName := stCntVw.stDataType.wsNameId :="bool";
ELSIF  stCnt.eDataType = E_DataType.eDataType_int THEN
	stCntVw.stDataType.wsName := stCntVw.stDataType.wsNameId :="int";
ELSIF  stCnt.eDataType = E_DataType.eDataType_lreal THEN
	stCntVw.stDataType.wsName := stCntVw.stDataType.wsNameId :="lreal";
ELSIF  stCnt.eDataType = E_DataType.eDataType_time_ms THEN
	stCntVw.stDataType.wsName := stCntVw.stDataType.wsNameId :="time_ms";
ELSIF  stCnt.eDataType = E_DataType.eDataType_time_s THEN
	stCntVw.stDataType.wsName := stCntVw.stDataType.wsNameId :="time_s";		
ELSIF  stCnt.eDataType = E_DataType.eDataType_wstring THEN
	stCntVw.stDataType.wsName := stCntVw.stDataType.wsNameId :="wstring";
END_IF

IF (stCnt.stName.wsName = "") AND (stCnt.stName.wsNameId = "")  THEN
	stCntVw.stUserLevel.wsName := "";		
ELSIF stCnt.eUserLevel = E_User_Level.eUser_Level_none THEN
	stCntVw.stUserLevel.wsName := stCntVw.stUserLevel.wsNameId := "none";
ELSIF stCnt.eUserLevel = E_User_Level.eUser_Level_Programmer THEN
	stCntVw.stUserLevel.wsName := stCntVw.stUserLevel.wsNameId := "programmer";				
ELSIF stCnt.eUserLevel = E_User_Level.eUser_Level_Admin THEN
	stCntVw.stUserLevel.wsName := stCntVw.stUserLevel.wsNameId := "admin";
ELSIF  stCnt.eUserLevel = E_User_Level.eUser_Level_Maintenance THEN
	stCntVw.stUserLevel.wsName := stCntVw.stUserLevel.wsNameId := "maintenance";
ELSIF  stCnt.eUserLevel = E_User_Level.eUser_Level_Manager THEN
	stCntVw.stUserLevel.wsName := stCntVw.stUserLevel.wsNameId := "manager";
ELSIF  stCnt.eUserLevel = E_User_Level.eUser_Level_Operator THEN
	stCntVw.stUserLevel.wsName := stCntVw.stUserLevel.wsNameId := "operator";
ELSIF  stCnt.eUserLevel = E_User_Level.eUser_Level_Level4 THEN
	stCntVw.stUserLevel.wsName := stCntVw.stUserLevel.wsNameId := "level4";
END_IF

IF (stCnt.stName.wsName = "") AND (stCnt.stName.wsNameId = "")  THEN
	RETURN;
END_IF	
	
stCntVw.stName := stCnt.stName;
stCntVw.stGroup := stCnt.stGroup;	
stCntVw.stValueOk.wsName := stCntVw.stValueOk.wsNameId := TO_WSTRING(stCnt.nValueOk);	
stCntVw.stValueNok.wsName := stCntVw.stValueNok.wsNameId := TO_WSTRING(stCnt.nValueNok);
stCntVw.stValueTotal.wsName := stCntVw.stValueTotal.wsNameId := TO_WSTRING(stCnt.nValueOk + stCnt.nValueNok);

stCntVw.stValueOkLevel1.wsName := stCntVw.stValueOkLevel1.wsNameId := TO_WSTRING(stCnt.nValueOkLevel1);
stCntVw.stValueNokLevel1.wsName := stCntVw.stValueNokLevel1.wsNameId := TO_WSTRING(stCnt.nValueNokLevel1);

stCntVw.stValueOkLevel2.wsName := stCntVw.stValueOkLevel2.wsNameId := TO_WSTRING(stCnt.nValueOkLevel2);
stCntVw.stValueNokLevel2.wsName := stCntVw.stValueNokLevel2.wsNameId := TO_WSTRING(stCnt.nValueNokLevel2);	

stCntVw.stValueTotalLevel1.wsName := stCntVw.stValueTotalLevel1.wsNameId := TO_WSTRING(stCnt.nValueTotalLevel1);
stCntVw.stValueTotalLevel2.wsName := stCntVw.stValueTotalLevel2.wsNameId := TO_WSTRING(stCnt.nValueTotalLevel2);			

	//reaction Ok level 1
IF (stCnt.eReactionOkLevel1 = E_CounterReaction.eCounterReaction_None) THEN
	stCntVw.stReactionOkLevel1.wsName := "none";					
ELSIF stCnt.eReactionOkLevel1 = E_CounterReaction.eCounterReaction_Info THEN
	stCntVw.stReactionOkLevel1.wsName:= stCntVw.stUserLevel.wsNameId := "info";			
ELSIF stCnt.eReactionOkLevel1 = E_CounterReaction.eCounterReaction_Warning THEN
	stCntVw.stReactionOkLevel1.wsName:= stCntVw.stUserLevel.wsNameId := "warning";
ELSIF stCnt.eReactionOkLevel1 = E_CounterReaction.eCounterReaction_Error THEN
	stCntVw.stReactionOkLevel1.wsName:= stCntVw.stUserLevel.wsNameId := "error";
ELSIF stCnt.eReactionOkLevel1 = E_CounterReaction.eCounterReaction_SerialFault_Warning THEN
	stCntVw.stReactionOkLevel1.wsName:= stCntVw.stUserLevel.wsNameId := "not used";
ELSIF stCnt.eReactionOkLevel1 = E_CounterReaction.eCounterReaction_SerialFault_Error THEN
	stCntVw.stReactionOkLevel1.wsName:= stCntVw.stUserLevel.wsNameId := "not used";		
END_IF	

//reaction Nok level 1
IF (stCnt.eReactionNokLevel1 = E_CounterReaction.eCounterReaction_None) THEN
	stCntVw.stReactionNokLevel1.wsName := "none";
ELSIF stCnt.eReactionNokLevel1 = E_CounterReaction.eCounterReaction_Info THEN
	stCntVw.stReactionNokLevel1.wsName:= stCntVw.stUserLevel.wsNameId := "info";			
ELSIF stCnt.eReactionNokLevel1 = E_CounterReaction.eCounterReaction_Warning THEN
	stCntVw.stReactionNokLevel1.wsName:= stCntVw.stUserLevel.wsNameId := "warning";
ELSIF stCnt.eReactionNokLevel1 = E_CounterReaction.eCounterReaction_Error THEN
	stCntVw.stReactionNokLevel1.wsName:= stCntVw.stUserLevel.wsNameId := "error";				
ELSIF stCnt.eReactionNokLevel1 = E_CounterReaction.eCounterReaction_SerialFault_Warning THEN
	stCntVw.stReactionNokLevel1.wsName:= stCntVw.stUserLevel.wsNameId := "serialfaultwarning";
ELSIF stCnt.eReactionNokLevel1 = E_CounterReaction.eCounterReaction_SerialFault_Error THEN
	stCntVw.stReactionNokLevel1.wsName:= stCntVw.stUserLevel.wsNameId := "serialfaulterror";
END_IF


//reaction Ok Level 2
IF (stCnt.eReactionOkLevel2 = E_CounterReaction.eCounterReaction_None) THEN
	stCntVw.stReactionOkLevel2.wsName := "none";					
ELSIF stCnt.eReactionOkLevel2 = E_CounterReaction.eCounterReaction_Info THEN
	stCntVw.stReactionOkLevel2.wsName:= stCntVw.stUserLevel.wsNameId := "info";			
ELSIF stCnt.eReactionOkLevel2 = E_CounterReaction.eCounterReaction_Warning THEN
	stCntVw.stReactionOkLevel2.wsName:= stCntVw.stUserLevel.wsNameId := "warning";
ELSIF stCnt.eReactionOkLevel2 = E_CounterReaction.eCounterReaction_Error THEN
	stCntVw.stReactionOkLevel2.wsName:= stCntVw.stUserLevel.wsNameId := "error";
ELSIF stCnt.eReactionOkLevel2 = E_CounterReaction.eCounterReaction_SerialFault_Warning THEN
	stCntVw.stReactionOkLevel2.wsName:= stCntVw.stUserLevel.wsNameId := "serialfaultwarning";
ELSIF stCnt.eReactionOkLevel2 = E_CounterReaction.eCounterReaction_SerialFault_Error THEN
	stCntVw.stReactionOkLevel2.wsName:= stCntVw.stUserLevel.wsNameId := "serialfaulterror";		
END_IF	

//reaction Nok Level 2
IF (stCnt.eReactionNokLevel2 = E_CounterReaction.eCounterReaction_None) THEN
	stCntVw.stReactionNokLevel2.wsName := "none";
ELSIF stCnt.eReactionNokLevel2 = E_CounterReaction.eCounterReaction_Info THEN
	stCntVw.stReactionNokLevel2.wsName:= stCntVw.stUserLevel.wsNameId := "info";			
ELSIF stCnt.eReactionNokLevel2 = E_CounterReaction.eCounterReaction_Warning THEN
	stCntVw.stReactionNokLevel2.wsName:= stCntVw.stUserLevel.wsNameId := "warning";
ELSIF stCnt.eReactionNokLevel2 = E_CounterReaction.eCounterReaction_Error THEN
	stCntVw.stReactionNokLevel2.wsName:= stCntVw.stUserLevel.wsNameId := "error";				
ELSIF stCnt.eReactionNokLevel2 = E_CounterReaction.eCounterReaction_SerialFault_Warning THEN
	stCntVw.stReactionNokLevel2.wsName:= stCntVw.stUserLevel.wsNameId := "serialfaultwarning";
ELSIF stCnt.eReactionNokLevel2 = E_CounterReaction.eCounterReaction_SerialFault_Error THEN
	stCntVw.stReactionNokLevel2.wsName:= stCntVw.stUserLevel.wsNameId := "serialfaulterror";
END_IF


//reaction total level 1
IF (stCnt.eReactionTotalLevel1 = E_CounterReaction.eCounterReaction_None) THEN
	stCntVw.stReactionTotalLevel1.wsName := "none";	
ELSIF stCnt.eReactionTotalLevel1 = E_CounterReaction.eCounterReaction_Info THEN
	stCntVw.stReactionTotalLevel1.wsName:= stCntVw.stUserLevel.wsNameId := "info";		
ELSIF stCnt.eReactionTotalLevel1 = E_CounterReaction.eCounterReaction_Warning THEN
	stCntVw.stReactionTotalLevel1.wsName:= stCntVw.stUserLevel.wsNameId := "warning";
ELSIF stCnt.eReactionTotalLevel1 = E_CounterReaction.eCounterReaction_Error THEN
	stCntVw.stReactionTotalLevel1.wsName:= stCntVw.stUserLevel.wsNameId := "error";				
ELSIF stCnt.eReactionTotalLevel1 = E_CounterReaction.eCounterReaction_SerialFault_Warning THEN
	stCntVw.stReactionTotalLevel1.wsName:= stCntVw.stUserLevel.wsNameId := "not used";
ELSIF stCnt.eReactionTotalLevel1 = E_CounterReaction.eCounterReaction_SerialFault_Error THEN
	stCntVw.stReactionTotalLevel1.wsName:= stCntVw.stUserLevel.wsNameId := "not used";

END_IF	

//reaction total level 2
IF (stCnt.eReactionTotalLevel2 = E_CounterReaction.eCounterReaction_None) THEN
	stCntVw.stReactionTotalLevel2.wsName := "none";	
ELSIF stCnt.eReactionTotalLevel2 = E_CounterReaction.eCounterReaction_Info THEN
	stCntVw.stReactionTotalLevel2.wsName:= stCntVw.stUserLevel.wsNameId := "info";	
ELSIF stCnt.eReactionTotalLevel2 = E_CounterReaction.eCounterReaction_Warning THEN
	stCntVw.stReactionTotalLevel2.wsName:= stCntVw.stUserLevel.wsNameId := "warning";
ELSIF stCnt.eReactionTotalLevel2 = E_CounterReaction.eCounterReaction_Error THEN
	stCntVw.stReactionTotalLevel2.wsName:= stCntVw.stUserLevel.wsNameId := "error";				
ELSIF stCnt.eReactionTotalLevel2 = E_CounterReaction.eCounterReaction_SerialFault_Warning THEN
	stCntVw.stReactionTotalLevel2.wsName:= stCntVw.stUserLevel.wsNameId := "not used";
ELSIF stCnt.eReactionTotalLevel2 = E_CounterReaction.eCounterReaction_SerialFault_Error THEN
	stCntVw.stReactionTotalLevel2.wsName:= stCntVw.stUserLevel.wsNameId := "not used";
END_IF

M_SetUpCounterViewTxt := TRUE;
END_METHOD

METHOD M_Supervision : ST_Text
VAR_INPUT
END_VAR
M_Supervision := F_CreateDynText("",0);
FOR ii := 0 TO CONST.iMaxIdxCounter DO

	stCounter[ii].nValueTotal := stCounter[ii].nValueOk + stCounter[ii].nValueNok;

	IF stCounter[ii].nValueOk >= stCounter[ii].eReactionOkLevel1 AND (stCounter[ii].eReactionOkLevel1 <> E_CounterReaction.eCounterReaction_None) THEN
		eSupervisionReaction := stCounter[ii].eReactionTotalLevel2;
		CASE stCounter[ii].eReactionOkLevel1 OF
			E_CounterReaction.eCounterReaction_Info:
				M_Supervision := F_CreateDynText(WCONCAT(stCounter[ii].stName.wsName," : Counter Reaction Ok Level 1 Info"),0);		
			E_CounterReaction.eCounterReaction_Warning:
				M_Supervision := F_CreateDynText(WCONCAT(stCounter[ii].stName.wsName,": Counter Reaction Ok Level 1 Warning"),0);		
			E_CounterReaction.eCounterReaction_Error:
				M_Supervision := F_CreateDynText(WCONCAT(stCounter[ii].stName.wsName,": Counter Reaction Ok Level 1 Error"),0);	
			E_CounterReaction.eCounterReaction_SerialFault_Warning:
				M_Supervision := F_CreateDynText(WCONCAT(stCounter[ii].stName.wsName,": Counter Reaction Ok Level 1 not aviable"),0);			
			E_CounterReaction.eCounterReaction_SerialFault_Error:
				M_Supervision := F_CreateDynText(WCONCAT(stCounter[ii].stName.wsName,": Counter Reaction Ok Level 1 not aviable"),0);			
		END_CASE	
	END_IF

	IF stCounter[ii].nValueOk >= stCounter[ii].eReactionOkLevel2 AND (stCounter[ii].eReactionOkLevel2 <> E_CounterReaction.eCounterReaction_None) THEN
		eSupervisionReaction := stCounter[ii].eReactionTotalLevel2;
		CASE stCounter[ii].eReactionOkLevel2 OF
			E_CounterReaction.eCounterReaction_Info:
				M_Supervision := F_CreateDynText(WCONCAT(stCounter[ii].stName.wsName," : Counter Reaction Ok Level 2 Info"),0);		
			E_CounterReaction.eCounterReaction_Warning:
				M_Supervision := F_CreateDynText(WCONCAT(stCounter[ii].stName.wsName,": Counter Reaction Ok Level 2 Warning"),0);		
			E_CounterReaction.eCounterReaction_Error:
				M_Supervision := F_CreateDynText(WCONCAT(stCounter[ii].stName.wsName,": Counter Reaction Ok Level 2 Error"),0);	
			E_CounterReaction.eCounterReaction_SerialFault_Warning:
				M_Supervision := F_CreateDynText(WCONCAT(stCounter[ii].stName.wsName,": Counter Reaction Ok Level 2 not aviable"),0);			
			E_CounterReaction.eCounterReaction_SerialFault_Error:
				M_Supervision := F_CreateDynText(WCONCAT(stCounter[ii].stName.wsName,": Counter Reaction Ok Level 2 not aviable"),0);			
		END_CASE	
	END_IF

	IF stCounter[ii].nValueNok >= stCounter[ii].eReactionNokLevel1 AND (stCounter[ii].eReactionNokLevel1 <> E_CounterReaction.eCounterReaction_None) THEN
		eSupervisionReaction := stCounter[ii].eReactionTotalLevel2;
		CASE stCounter[ii].eReactionNokLevel1 OF
			E_CounterReaction.eCounterReaction_Info:
				M_Supervision := F_CreateDynText(WCONCAT(stCounter[ii].stName.wsName," : Counter Reaction Nok Level 1 Info"),0);		
			E_CounterReaction.eCounterReaction_Warning:
				M_Supervision := F_CreateDynText(WCONCAT(stCounter[ii].stName.wsName,": Counter Reaction Nok Level 1 Warning"),0);		
			E_CounterReaction.eCounterReaction_Error:
				M_Supervision := F_CreateDynText(WCONCAT(stCounter[ii].stName.wsName,": Counter Reaction Nok Level 1 Error"),0);	
			E_CounterReaction.eCounterReaction_SerialFault_Warning:
				M_Supervision := F_CreateDynText(WCONCAT(stCounter[ii].stName.wsName,": Counter Reaction Nok Level 1 Serial Warning"),0);			
			E_CounterReaction.eCounterReaction_SerialFault_Error:
				M_Supervision := F_CreateDynText(WCONCAT(stCounter[ii].stName.wsName,": Counter Reaction Nok Level 1 Serial Warning Stop"),0);			
		END_CASE	
	END_IF

	IF stCounter[ii].nValueNok >= stCounter[ii].eReactionNokLevel2 AND (stCounter[ii].eReactionNokLevel2 <> E_CounterReaction.eCounterReaction_None) THEN
		eSupervisionReaction := stCounter[ii].eReactionTotalLevel2;
		CASE stCounter[ii].eReactionNokLevel2 OF
			E_CounterReaction.eCounterReaction_Info:
				M_Supervision := F_CreateDynText(WCONCAT(stCounter[ii].stName.wsName," : Counter Reaction Nok Level 2 Info"),0);		
			E_CounterReaction.eCounterReaction_Warning:
				M_Supervision := F_CreateDynText(WCONCAT(stCounter[ii].stName.wsName,": Counter Reaction Nok Level 2 Warning"),0);		
			E_CounterReaction.eCounterReaction_Error:
				M_Supervision := F_CreateDynText(WCONCAT(stCounter[ii].stName.wsName,": Counter Reaction Nok Level 2 Error"),0);	
			E_CounterReaction.eCounterReaction_SerialFault_Warning:
				M_Supervision := F_CreateDynText(WCONCAT(stCounter[ii].stName.wsName,": Counter Reaction Nok Level 2 Serial Warning"),0);			
			E_CounterReaction.eCounterReaction_SerialFault_Error:
				M_Supervision := F_CreateDynText(WCONCAT(stCounter[ii].stName.wsName,": Counter Reaction Nok Level 2 Serial Warning Stop"),0);			
		END_CASE	
	END_IF	
	
	IF stCounter[ii].nValueTotal >= stCounter[ii].eReactionTotalLevel1 AND (stCounter[ii].eReactionTotalLevel1 <> E_CounterReaction.eCounterReaction_None) THEN
		eSupervisionReaction := stCounter[ii].eReactionTotalLevel2;
		CASE stCounter[ii].eReactionTotalLevel1 OF
			E_CounterReaction.eCounterReaction_Info:
				M_Supervision := F_CreateDynText(WCONCAT(stCounter[ii].stName.wsName," : Counter Reaction Total Level 1 Info"),0);		
			E_CounterReaction.eCounterReaction_Warning:
				M_Supervision := F_CreateDynText(WCONCAT(stCounter[ii].stName.wsName,": Counter Reaction Total Level 1 Warning"),0);		
			E_CounterReaction.eCounterReaction_Error:
				M_Supervision := F_CreateDynText(WCONCAT(stCounter[ii].stName.wsName,": Counter Reaction Total Level 1 Error"),0);	
			E_CounterReaction.eCounterReaction_SerialFault_Warning:
				M_Supervision := F_CreateDynText(WCONCAT(stCounter[ii].stName.wsName,": Counter Reaction Total Level 1 not aviable"),0);			
			E_CounterReaction.eCounterReaction_SerialFault_Error:
				M_Supervision := F_CreateDynText(WCONCAT(stCounter[ii].stName.wsName,": Counter Reaction Total Level 1 not aviable"),0);			
		END_CASE	
	END_IF
	IF stCounter[ii].nValueTotal >= stCounter[ii].eReactionTotalLevel2 AND (stCounter[ii].eReactionTotalLevel2 <> E_CounterReaction.eCounterReaction_None) THEN
		eSupervisionReaction := stCounter[ii].eReactionTotalLevel2;
		CASE stCounter[ii].eReactionTotalLevel2 OF
			E_CounterReaction.eCounterReaction_Info:
				M_Supervision := F_CreateDynText(WCONCAT(stCounter[ii].stName.wsName," : Counter Reaction Total Level 2 Info"),0);		
			E_CounterReaction.eCounterReaction_Warning:
				M_Supervision := F_CreateDynText(WCONCAT(stCounter[ii].stName.wsName,": Counter Reaction Total Level 2 Warning"),0);		
			E_CounterReaction.eCounterReaction_Error:
				M_Supervision := F_CreateDynText(WCONCAT(stCounter[ii].stName.wsName,": Counter Reaction Total Level 2 Error"),0);	
			E_CounterReaction.eCounterReaction_SerialFault_Warning:
				M_Supervision := F_CreateDynText(WCONCAT(stCounter[ii].stName.wsName,": Counter Reaction Total Level 2 not aviable"),0);			
			E_CounterReaction.eCounterReaction_SerialFault_Error:
				M_Supervision := F_CreateDynText(WCONCAT(stCounter[ii].stName.wsName,": Counter Reaction Total Level 2 not aviable"),0);			
		END_CASE	
	END_IF
END_FOR
END_METHOD

END_FUNCTION_BLOCK

// ---- POUs/Safety/TwinSAFE_Diagnose/FB_TwinSAFEDiag_EmergencyStop.TcPOU
FUNCTION_BLOCK FB_TwinSAFEDiag_EmergencyStop
VAR_INPUT
	wsFunctionBlockText		: WSTRING;
	stIn					: ST_SafetyDiagInfo;
END_VAR
VAR_OUTPUT
	bError					: BOOL;
	stErrorText				: ST_Text;
	stErrorTextAdd			: ST_Text;
END_VAR
VAR
	{attribute 'hide' := ''}
	wsTempText: WSTRING(255);
END_VAR

bError := FALSE;
stErrorText := stEmptyText;
stErrorTextAdd := stEmptyText;

(*	DIAG:
	Bit 0: Disc Error (EStopIn1/2)
	Bit 1: Disc Error (EStopIn3/4)
	Bit 2: Disc Error (EStopIn5/6)
	Bit 3: Disc Error (EStopIn7/8)
	Bit 4: EDM1 Error
	Bit 5: EDM2 Error		*)
IF stIn.uintDiag.0 THEN
	bError := TRUE;
	stErrorText := stTextListGlobal.stText_Safety.stText_Safety_Discrepancy_Error;
	wsTempText := (WCONCAT(WCONCAT(wsFunctionBlockText, "; ") , "Channel: 1/2"));
	stErrorTextAdd := F_CreateDynTextDefault(wsTempText);

ELSIF stIn.uintDiag.1 THEN
	bError := TRUE;
	stErrorText := stTextListGlobal.stText_Safety.stText_Safety_Discrepancy_Error;
	wsTempText := (WCONCAT(WCONCAT(wsFunctionBlockText, "; ") , "Channel: 3/4"));
	stErrorTextAdd := F_CreateDynTextDefault(wsTempText);

ELSIF stIn.uintDiag.2 THEN
	bError := TRUE;
	stErrorText := stTextListGlobal.stText_Safety.stText_Safety_Discrepancy_Error;
	wsTempText := (WCONCAT(WCONCAT(wsFunctionBlockText, "; ") , "Channel: 5/6"));
	stErrorTextAdd := F_CreateDynTextDefault(wsTempText);

ELSIF stIn.uintDiag.3 THEN
	bError := TRUE;
	stErrorText := stTextListGlobal.stText_Safety.stText_Safety_Discrepancy_Error;
	wsTempText := (WCONCAT(WCONCAT(wsFunctionBlockText, "; ") , "Channel: 7/8"));
	stErrorTextAdd := F_CreateDynTextDefault(wsTempText);

ELSIF stIn.uintDiag.4 THEN
	bError := TRUE;
	stErrorText := stTextListGlobal.stText_Safety.stText_Safety_EDM_Error;
	wsTempText := (WCONCAT(WCONCAT(wsFunctionBlockText, "; ") , "EDM 1"));
	stErrorTextAdd := F_CreateDynTextDefault(wsTempText);

ELSIF stIn.uintDiag.5 THEN
	bError := TRUE;
	stErrorText := stTextListGlobal.stText_Safety.stText_Safety_EDM_Error;
	wsTempText := (WCONCAT(WCONCAT(wsFunctionBlockText, "; ") , "EDM 2"));
	stErrorTextAdd := F_CreateDynTextDefault(wsTempText);

(*	STATE
	1: State RUN
	2: State STOP
	3: State SAFE
	4: State ERROR
	5: State RESET
	6: State START
	8: State DELAYOUT	*)
ELSIF stIn.usintState = 4 THEN
	bError := TRUE;
	stErrorText := stTextListGlobal.stText_UnknownError;
	stErrorTextAdd := F_CreateDynTextDefault(wsFunctionBlockText);
END_IF

END_FUNCTION_BLOCK

// ---- POUs/Safety/TwinSAFE_Diagnose/FB_TwinSAFEDiag_MachineMonitoring.TcPOU
FUNCTION_BLOCK FB_TwinSAFEDiag_MachineMonitoring
VAR_INPUT
	wsFunctionBlockText		: WSTRING;
	stIn					AT %I*		: ST_SafetyDiagInfo;
END_VAR
VAR_OUTPUT
	bError					: BOOL;
	stErrorText				: ST_Text;
	stErrorTextAdd			: ST_Text;
END_VAR
VAR
	{attribute 'hide' := ''}
	wsTempText: WSTRING(255);
END_VAR

bError := FALSE;
stErrorText := stEmptyText;
stErrorTextAdd := stEmptyText;

(*	DIAG:
	Bit 0: Disc Error (MonIn1/2)
	Bit 1: Disc Error (Secure1/2)
	Bit 2: Disc Error (MonIn3/4)
	Bit 4: EDM1 Error
	Bit 5: EDM2 Error		*)
IF stIn.uintDiag.0 THEN
	bError := TRUE;
	stErrorText := stTextListGlobal.stText_Safety.stText_Safety_Discrepancy_Error;
	wsTempText := (WCONCAT(WCONCAT(wsFunctionBlockText, "; ") , "Channel: 1/2"));
	stErrorTextAdd := F_CreateDynTextDefault(wsTempText);

ELSIF stIn.uintDiag.1 THEN
	bError := TRUE;
	stErrorText := stTextListGlobal.stText_Safety.stText_Safety_Discrepancy_Error;
	wsTempText := (WCONCAT(WCONCAT(wsFunctionBlockText, "; ") , "Channel: Secure 1/2"));
	stErrorTextAdd := F_CreateDynTextDefault(wsTempText);

ELSIF stIn.uintDiag.2 THEN
	bError := TRUE;	
	stErrorText := stTextListGlobal.stText_Safety.stText_Safety_Discrepancy_Error;
	wsTempText := (WCONCAT(WCONCAT(wsFunctionBlockText, "; ") , "Channel: 3/4"));
	stErrorTextAdd := F_CreateDynTextDefault(wsTempText);

ELSIF stIn.uintDiag.4 THEN
	bError := TRUE;
	stErrorText := stTextListGlobal.stText_Safety.stText_Safety_EDM_Error;
	wsTempText := (WCONCAT(WCONCAT(wsFunctionBlockText, "; ") , "EDM 1"));
	stErrorTextAdd := F_CreateDynTextDefault(wsTempText);

ELSIF stIn.uintDiag.5 THEN
	bError := TRUE;
	stErrorText := stTextListGlobal.stText_Safety.stText_Safety_EDM_Error;
	wsTempText := (WCONCAT(WCONCAT(wsFunctionBlockText, "; ") , "EDM 2"));
	stErrorTextAdd := F_CreateDynTextDefault(wsTempText);

(*	STATE
	1: State RUN
	2: State STOP
	3: State SAFE
	4: State ERROR
	5: State RESET
	6: State START
	7: State ERRORDELAY
	8: State DELAYOUT
	9: State FUNCTEST	*)
ELSIF stIn.usintState = 4 THEN
	bError := TRUE;
	stErrorText := stTextListGlobal.stText_UnknownError;
	stErrorTextAdd := F_CreateDynTextDefault(wsFunctionBlockText);
END_IF

END_FUNCTION_BLOCK

// ---- POUs/Safety/TwinSAFE_Diagnose/FB_TwinSAFEDiag_TwoHand.TcPOU
FUNCTION_BLOCK FB_TwinSAFEDiag_TwoHand
VAR_INPUT
	wsFunctionBlockText	: WSTRING;
	stIn				: ST_SafetyDiagInfo;
END_VAR
VAR_OUTPUT
	bWarning: BOOL;	
	stWarningText: ST_Text;
	stWarningTextAdd: ST_Text;
	
	bError					: BOOL;
	stErrorText				: ST_Text;
	stErrorTextAdd			: ST_Text;
END_VAR
VAR
	{attribute 'hide' := ''}
	wsTempText: WSTRING(255);
END_VAR

bWarning := FALSE;
stWarningText := stEmptyText;
stWarningTextAdd := stEmptyText;

bError := FALSE;
stErrorText := stEmptyText;
stErrorTextAdd := stEmptyText;

(*	DIAG:
	Bit 0: Disc Error (TwoHand1/2)
	Bit 1: Disc Error (TwoHand3/4)
	Bit 2: Disc Error (InGroup1/2)
	Bit 6: TwoHand Error		*)
IF stIn.uintDiag.0 THEN
	bError := TRUE;
	stErrorText := stTextListGlobal.stText_Safety.stText_Safety_Discrepancy_Error;
	wsTempText := (WCONCAT(WCONCAT(wsFunctionBlockText, "; ") , "Channel: 1/2"));
	stErrorTextAdd := F_CreateDynTextDefault(wsTempText);

ELSIF stIn.uintDiag.1 THEN
	bError := TRUE;
	stErrorText := stTextListGlobal.stText_Safety.stText_Safety_Discrepancy_Error;
	wsTempText := (WCONCAT(WCONCAT(wsFunctionBlockText, "; ") , "Channel: 3/4"));
	stErrorTextAdd := F_CreateDynTextDefault(wsTempText);

ELSIF stIn.uintDiag.2 THEN
	bError := TRUE;
	stErrorText := stTextListGlobal.stText_Safety.stText_Safety_Discrepancy_Error;
	wsTempText := (WCONCAT(WCONCAT(wsFunctionBlockText, "; ") , "Group: 1/2"));
	stErrorTextAdd := F_CreateDynTextDefault(wsTempText);

ELSIF stIn.uintDiag.6 THEN
	bError := TRUE;
	stErrorText := stTextListGlobal.stText_Safety.stText_Safety_2Hand_Error;
	stErrorTextAdd := F_CreateDynTextDefault(wsTempText);

(*	STATE
	1: State RUN
	2: State STOP
	3: State SAFE
	4: State ERROR
	5: State RESET
	11: State 1BUTTON
	12: State 2BUTTON
	13: State RELEASE
	*)
ELSIF stIn.usintState = 4 THEN
	bError := TRUE;
	stErrorText := stTextListGlobal.stText_UnknownError;
	stErrorTextAdd := F_CreateDynTextDefault(wsFunctionBlockText);

END_IF

(*	Warnung		*)
IF stIn.usintState = 13 THEN
	bWarning := TRUE;
	stWarningText := stTextListGlobal.stText_Safety.stText_Safety_Discrepancy_Warning;
	stWarningTextAdd := F_CreateDynTextDefault(wsFunctionBlockText);
END_IF

END_FUNCTION_BLOCK

// ---- POUs/Safety/TwinSAFE_Diagnose/FB_TwinSAFEDiag_EDM.TcPOU
{attribute 'hide_all_locals'}
FUNCTION_BLOCK FB_TwinSAFEDiag_EDM
VAR_INPUT
	wsFunctionBlockText		: WSTRING;
	stIn					: ST_SafetyDiagInfo;
END_VAR
VAR_OUTPUT
	bError					: BOOL;
	stErrorText				: ST_Text;
	stErrorTextAdd			: ST_Text;
END_VAR

// Reset 
bError := FALSE;
stErrorText := stEmptyText;
stErrorTextAdd := stEmptyText;

(*	DIAG:
	Bit 0: Switch OFF Timer Timeout
	Bit 1: Switch ON Timer Timeout	*)
IF stIn.uintDiag.0 THEN
	bError := TRUE;
	stErrorText := stTextListGlobal.stText_Safety.stText_Safety_TimerSwitchOffTimeout;
	stErrorTextAdd := F_CreateDynTextDefault(wsFunctionBlockText);

ELSIF stIn.uintDiag.1 THEN
	bError := TRUE;
	stErrorText := stTextListGlobal.stText_Safety.stText_Safety_TimerSwitchOnTimeout;
	stErrorTextAdd := F_CreateDynTextDefault(wsFunctionBlockText);
(*	STATE
	2: State STOP
	4: State ERROR
	5: State RESET
	14: State MON_OFF
	15: State MON_ON	*)
ELSIF stIn.uintDiag = 4 THEN
	bError := TRUE;
	stErrorText := stTextListGlobal.stText_UnknownError;
	stErrorTextAdd := F_CreateDynTextDefault(wsFunctionBlockText);
END_IF

END_FUNCTION_BLOCK

// ---- POUs/Safety/TwinSAFE_Diagnose/FB_TwinSAFE_HW_Diag.TcPOU
/// diagnose from TwinSAFE hardware
{attribute 'hide_all_locals' := ''}
FUNCTION_BLOCK FB_TwinSAFE_HW_Diag
VAR_INPUT
	/// enable the function block
	bEnable: BOOL;
	/// EC master AMS adress
	stEcMasterAmsAdr: ST_AmsAddr;
	/// EC master device ID
	nEcMasterDevId: UINT;
	/// EC master device state
	nDeviceState: UINT;
	/// current system time
	dtNow: DT;
END_VAR
VAR_OUTPUT
	bError,
	bWarning			: BOOL;	
	stWarningText,
	stWarningTextAdd,
	
	stErrorText,
	stErrorTextAdd		: ST_Text;
END_VAR
VAR CONSTANT
	{attribute 'hide' := ''}
	nMAX_DiagSlaveSize: INT := 2000;
	{attribute 'hide' := ''}
	nMAX_HistoryDevice: INT := 100;
END_VAR
VAR
	/// AmsNetId of the EtherCAT master device 
	{attribute 'hide' := ''}
	sEcMasterNetId: T_AmsNetId;
	{attribute 'hide' := ''}
	fbEcGetAllSlaveAddr: FB_EcGetAllSlaveAddr;
	{attribute 'hide' := ''}
	fbEcGetSlaveIdentity: FB_EcGetSlaveIdentity;
	///	CoE		
	{attribute 'hide' := ''}
	fbEcCoeSdoRead: FB_EcCoESdoRead;
	/// CoE - Diag History
	{attribute 'hide' := ''}
	fbHistoryDiag: FB_Diagnosis_History;
	{attribute 'hide' := ''}
	sErrorTextTemp: T_MAXSTRING;
	///Get slave name
	{attribute 'hide' := ''}
	fbGetSlaveName: IOF_GetBoxNameByAddr;
	{attribute 'hide' := ''}
	nStep: INT;
	{attribute 'hide' := ''}
	tonStartUp: TON;
	{attribute 'hide' := ''}
	tonCycle: TON;
	{attribute 'hide' := ''}
	tonDelay: TON;
	{attribute 'hide' := ''}
	arrSlaves: ARRAY[0..nMAX_DiagSlaveSize] OF UINT;
	{attribute 'hide' := ''}
	arrSlaveIdent: ARRAY[0..nMAX_DiagSlaveSize] OF ST_EcSlaveIdentity;
	{attribute 'hide' := ''}
	arrSlaveType: ARRAY[0..nMAX_DiagSlaveSize] OF STRING;
	{attribute 'hide' := ''}
	aDiagHistoryMirror: ARRAY[0..nMAX_HistoryDevice] OF ST_DiagHistory;
	{attribute 'hide' := ''}
	nIdx: INT;
	{attribute 'hide' := ''}
	nHistoryDevice: INT;
	{attribute 'hide' := ''}
	nCoE_DiagDataA: WORD;
	{attribute 'hide' := ''}
	nCoE_DiagDataB: WORD;
	{attribute 'hide' := ''}
	nCoE_DiagDataC: WORD;
	{attribute 'hide' := ''}
	nCoE_DiagDataD: WORD;
	{attribute 'hide' := ''}
	nCoE_DiagDataE: WORD;
	{attribute 'hide' := ''}
	sErrorBoxame: STRING;
	{attribute 'hide' := ''}
	wsTempText: WSTRING(255);
END_VAR

(* Supported Hardware:
		EL1904
		EL1918
		EL2904
		EL2912
*)

(*	EtherCAT Master NetId	*)
sEcMasterNetId := F_CreateAmsNetId(nIds := stEcMasterAmsAdr.netId);

tonStartUp(IN := bEnable AND nDeviceState = 0, PT := T#2S);
tonDelay(PT := T#100MS);
tonDelay.IN := FALSE;

CASE nStep OF

	0:
		IF tonStartUp.Q THEN
			fbEcGetAllSlaveAddr(sNetId:= sEcMasterNetId ,
							pAddrBuf:= ADR(arrSlaves),
							cbBufLen:= SIZEOF(arrSlaves),
							bExecute:= FALSE );
			nIdx := 0;
			nHistoryDevice := 0;
			
			M_Reset();
			nStep := 10;
		END_IF

(*	Get all slaves identities	*)
	10..299:
		M_GetSlaveIdentity();
	
(*	read out status	*)
	300..399:
		// EL1904 and EL2904
		M_GetState_ErrorNumber();
	
	400..499:
		// EL1918 and EL2912
		M_GetState_History();


(*	Detail Diagnose	*)
	600..699:
		M_DiagnosisAlarm();

(*	ERROR	*)

		(*	neuer Versuch	*)
	1000:
		tonCycle( IN := bEnable , PT := T#30s);
		IF tonCycle.Q THEN
			tonCycle( IN := FALSE , PT := T#5s);
			nStep := 0;
		END_IF

END_CASE

/// diagnose device and raise alarm 
METHOD PRIVATE M_DiagnosisAlarm : BOOL
CASE nStep OF
	600:
		fbGetSlaveName(NETID		:= '',	(*local*)
						DEVICEID	:= nEcMasterDevId,
						BOXADDR		:= arrSlaves[nIdx],
						START		:= FALSE);
		IF NOT fbGetSlaveName.Busy THEN
			nStep := 610;
		END_IF

	610:
		fbGetSlaveName(NETID		:= '',	(*local*)
						DEVICEID	:= nEcMasterDevId,
						BOXADDR		:= arrSlaves[nIdx],
						START		:= TRUE);
		IF fbGetSlaveName.Busy AND NOT fbGetSlaveName.ERR THEN
			nStep := 612;
		ELSIF fbGetSlaveName.ERR THEN
			nStep := 1000;
		END_IF

	612:
		fbGetSlaveName(NETID		:= '',	(*local*)
						DEVICEID	:= nEcMasterDevId,
						BOXADDR		:= arrSlaves[nIdx],
						START		:= TRUE);
		IF NOT fbGetSlaveName.Busy AND NOT fbGetSlaveName.ERR THEN
			sErrorBoxame := fbGetSlaveName.BOXNAME;
			nStep := 620;
		ELSIF fbGetSlaveName.ERR THEN
			bWarning := TRUE;
			stWarningText := stTextListGlobal.stText_EcGetSlaveNameErr;
			wsTempText := WCONCAT("ErrId: ", UDINT_TO_WSTRING(fbGetSlaveName.ERRID));
			wsTempText := WCONCAT(wsTempText, "; SlaveNb: ");
			wsTempText := WCONCAT(wsTempText, UINT_TO_WSTRING(arrSlaves[nIdx]));
			stWarningTextAdd := F_CreateDynTextDefault(wsTempText);
			nStep := 1000;
		END_IF

	620:
		fbGetSlaveName(NETID		:= '',	(*local*)
						DEVICEID	:= nEcMasterDevId,
						BOXADDR		:= arrSlaves[nIdx],
						START		:= FALSE);
		IF NOT fbGetSlaveName.Busy THEN
			nStep := 630;
		END_IF

	630: // create error message
		bError := TRUE;
		stErrorText := stTextListGlobal.stText_Safety.stText_Safety_Error_Diagnosis;
		wsTempText := WCONCAT("Slave: ", TO_WSTRING(sErrorBoxame));
		IF LEFT(arrSlaveType[nIdx] , 6) = 'EL1904' THEN
			stErrorText := stTextListGlobal.stText_Safety.stText_Safety_Error_SensortestInput;
			IF nCoE_DiagDataA.0 THEN				
				wsTempText := WCONCAT(wsTempText, "; Input: 1");
			ELSIF nCoE_DiagDataA.1 THEN
				wsTempText := WCONCAT(wsTempText, "; Input: 2");
			ELSIF nCoE_DiagDataA.2 THEN
				wsTempText := WCONCAT(wsTempText, "; Input: 3");
			ELSIF nCoE_DiagDataA.3 THEN
				wsTempText := WCONCAT(wsTempText, "; Input: 4");

			ELSIF nCoE_DiagDataB.0 THEN
				stErrorText := stTextListGlobal.stText_Safety.stText_Safety_Error_FirstInputPair;
			ELSIF nCoE_DiagDataB.1 THEN
				stErrorText := stTextListGlobal.stText_Safety.stText_Safety_Error_SecondInputPair;
			END_IF			

		ELSIF LEFT(arrSlaveType[nIdx] , 6) = 'EL2904' THEN
			IF nCoE_DiagDataC.0 OR nCoE_DiagDataC.4 THEN
					wsTempText := WCONCAT(wsTempText, "; Output: 1");
				IF nCoE_DiagDataC.1 OR nCoE_DiagDataC.5 THEN
					wsTempText := WCONCAT(wsTempText, "; Output: 2");
				ELSIF nCoE_DiagDataC.2 OR nCoE_DiagDataC.6 THEN
					wsTempText := WCONCAT(wsTempText, "; Output: 3");
				ELSIF nCoE_DiagDataC.3 OR nCoE_DiagDataC.7 THEN
					wsTempText := WCONCAT(wsTempText, "; Output: 4");
				END_IF
			END_IF
			
